C01814=1167.617,49.371,-49.076,-179.587,6.107,148.976
C01815=1167.621,49.121,-49.060,-179.589,6.107,148.977
C01816=1167.627,48.872,-49.044,-179.592,6.106,148.978
C01817=1167.632,48.622,-49.029,-179.594,6.104,148.978
C01818=1167.636,48.373,-49.012,-179.597,6.104,148.979
C01819=1167.641,48.124,-48.997,-179.599,6.103,148.979
C01820=1167.647,47.874,-48.981,-179.602,6.102,148.980
C01821=1167.652,47.624,-48.965,-179.605,6.101,148.980
C01822=1167.656,47.375,-48.950,-179.607,6.100,148.981
C01823=1167.662,47.126,-48.935,-179.610,6.099,148.982
C01824=1167.666,46.876,-48.919,-179.612,6.098,148.982
C01825=1167.671,46.627,-48.902,-179.615,6.098,148.983
C01826=1167.677,46.377,-48.887,-179.618,6.096,148.983
C01827=1167.681,46.128,-48.872,-179.621,6.096,148.984
C01828=1167.686,45.878,-48.856,-179.623,6.095,148.984
C01829=1167.692,45.629,-48.840,-179.626,6.093,148.985
C01830=1167.696,45.380,-48.825,-179.628,6.093,148.985
C01831=1167.702,45.130,-48.810,-179.631,6.092,148.986
C01832=1167.706,44.880,-48.794,-179.633,6.090,148.986
C01833=1167.712,44.631,-48.778,-179.636,6.090,148.987
C01834=1167.716,44.382,-48.763,-179.638,6.089,148.988
C01835=1167.721,44.132,-48.747,-179.641,6.088,148.988
C01836=1167.727,43.882,-48.732,-179.644,6.087,148.989
C01837=1167.731,43.633,-48.717,-179.646,6.086,148.989
C01838=1167.737,43.384,-48.701,-179.648,6.085,148.990
C01839=1167.742,43.134,-48.686,-179.652,6.084,148.990
C01840=1167.746,42.884,-48.670,-179.654,6.083,148.991
C01841=1167.752,42.635,-48.655,-179.656,6.083,148.992
C01842=1167.757,42.386,-48.639,-179.660,6.082,148.992
C01843=1167.762,42.137,-48.624,-179.662,6.081,148.993
C01844=1167.766,41.886,-48.608,-179.664,6.080,148.993
C01845=1167.771,41.637,-48.593,-179.667,6.079,148.994
C01846=1167.776,41.388,-48.577,-179.670,6.078,148.994
C01847=1167.782,41.139,-48.562,-179.672,6.077,148.995
C01848=1167.787,40.889,-48.548,-179.675,6.077,148.996
C01849=1167.792,40.639,-48.532,-179.677,6.075,148.996
C01850=1167.797,40.389,-48.516,-179.680,6.075,148.997
C01851=1167.802,40.140,-48.501,-179.682,6.074,148.997
C01852=1167.807,39.891,-48.485,-179.685,6.072,148.998
C01853=1167.812,39.642,-48.470,-179.688,6.072,148.998
C01854=1167.817,39.392,-48.455,-179.690,6.071,148.999
C01855=1167.822,39.143,-48.441,-179.693,6.071,149.000
C01856=1167.827,38.893,-48.425,-179.696,6.069,149.000
C01857=1167.832,38.643,-48.409,-179.698,6.068,149.001
C01858=1167.837,38.394,-48.394,-179.700,6.068,149.001
C01859=1167.842,38.145,-48.379,-179.703,6.067,149.002
C01860=1167.847,37.895,-48.364,-179.706,6.065,149.002
C01861=1167.852,37.646,-48.349,-179.708,6.065,149.003
C01862=1167.857,37.396,-48.334,-179.711,6.064,149.003
C01863=1167.862,37.146,-48.318,-179.714,6.063,149.004
C01864=1167.867,36.897,-48.303,-179.716,6.062,149.005
C01865=1167.872,36.647,-48.288,-179.719,6.061,149.005
C01866=1167.877,36.398,-48.273,-179.721,6.061,149.006
C01867=1167.882,36.149,-48.257,-179.724,6.059,149.006
C01868=1167.887,35.899,-48.243,-179.727,6.059,149.007
C01869=1167.893,35.650,-48.227,-179.729,6.058,149.007
C01870=1167.897,35.401,-48.212,-179.732,6.057,149.008
C01871=1167.903,35.151,-48.197,-179.734,6.056,149.009
C01872=1167.907,34.901,-48.182,-179.737,6.055,149.009
C01873=1167.912,34.651,-48.167,-179.739,6.054,149.010
C01874=1167.917,34.402,-48.152,-179.742,6.054,149.010
C01875=1167.922,34.153,-48.137,-179.745,6.053,149.011
C01876=1167.927,33.903,-48.122,-179.747,6.052,149.012
C01877=1167.932,33.653,-48.107,-179.750,6.051,149.012
C01878=1167.938,33.404,-48.092,-179.752,6.050,149.013
C01879=1167.942,33.155,-48.077,-179.755,6.049,149.013
C01880=1167.948,32.905,-48.062,-179.757,6.048,149.014
C01881=1167.953,32.656,-48.047,-179.760,6.048,149.014
C01882=1167.958,32.406,-48.033,-179.762,6.047,149.015
C01883=1167.963,32.157,-48.017,-179.765,6.046,149.016
C01884=1167.968,31.908,-48.002,-179.768,6.045,149.016
C01885=1167.973,31.658,-47.988,-179.770,6.044,149.017
C01886=1167.978,31.408,-47.972,-179.773,6.044,149.017
C01887=1167.983,31.159,-47.958,-179.775,6.043,149.018
C01888=1167.988,30.909,-47.942,-179.778,6.042,149.018
C01889=1167.993,30.660,-47.928,-179.780,6.041,149.019
C01890=1167.998,30.411,-47.913,-179.783,6.040,149.020
C01891=1168.004,30.161,-47.898,-179.785,6.040,149.020
C01892=1168.008,29.911,-47.883,-179.788,6.038,149.021
C01893=1168.013,29.662,-47.869,-179.791,6.038,149.021
C01894=1168.019,29.412,-47.853,-179.793,6.037,149.022
C01895=1168.024,29.163,-47.839,-179.796,6.036,149.023
C01896=1168.028,28.914,-47.824,-179.798,6.036,149.023
C01897=1168.033,28.664,-47.810,-179.801,6.034,149.024
C01898=1168.039,28.395,-47.794,-179.804,6.034,149.024
C01899=1168.044,28.126,-47.778,-179.806,6.033,149.025
C01900=1168.050,27.857,-47.762,-179.809,6.032,149.025
C01901=1168.055,27.588,-47.746,-179.812,6.031,149.026
C01902=1168.060,27.339,-47.731,-179.814,6.030,149.027
C01903=1168.065,27.089,-47.717,-179.817,6.029,149.027
C01904=1168.071,26.839,-47.702,-179.820,6.029,149.028
C01905=1168.075,26.590,-47.687,-179.822,6.028,149.028
C01906=1168.080,26.340,-47.672,-179.825,6.027,149.029
C01907=1168.085,26.091,-47.657,-179.827,6.026,149.030
C01908=1168.090,25.841,-47.643,-179.830,6.025,149.030
C01909=1168.095,25.592,-47.628,-179.832,6.024,149.031
C01910=1168.100,25.342,-47.613,-179.835,6.024,149.031
C01911=1168.105,25.093,-47.599,-179.838,6.023,149.032
C01912=1168.111,24.843,-47.584,-179.840,6.023,149.033
C01913=1168.116,24.594,-47.570,-179.843,6.021,149.033
C01914=1168.121,24.345,-47.555,-179.845,6.020,149.034
C01915=1168.126,24.095,-47.541,-179.848,6.020,149.034
C01916=1168.131,23.845,-47.527,-179.850,6.019,149.035
C01917=1168.135,23.596,-47.512,-179.853,6.019,149.035
C01918=1168.141,23.346,-47.497,-179.856,6.017,149.036
C01919=1168.146,23.096,-47.483,-179.858,6.016,149.037
C01920=1168.151,22.847,-47.468,-179.861,6.016,149.037
C01921=1168.156,22.598,-47.453,-179.863,6.015,149.038
C01922=1168.161,22.348,-47.439,-179.866,6.015,149.038
C01923=1168.166,22.099,-47.425,-179.868,6.014,149.039
C01924=1168.171,21.849,-47.411,-179.871,6.013,149.040
C01925=1168.177,21.600,-47.395,-179.874,6.012,149.040
C01926=1168.182,21.350,-47.381,-179.876,6.011,149.041
C01927=1168.186,21.100,-47.367,-179.878,6.011,149.041
C01928=1168.191,20.851,-47.352,-179.881,6.010,149.042
C01929=1168.196,20.601,-47.338,-179.883,6.009,149.042
C01930=1168.201,20.351,-47.324,-179.886,6.008,149.043
C01931=1168.207,20.103,-47.309,-179.889,6.007,149.044
C01932=1168.212,19.853,-47.295,-179.891,6.007,149.044
C01933=1168.217,19.603,-47.281,-179.893,6.006,149.045
C01934=1168.221,19.354,-47.266,-179.896,6.006,149.045
C01935=1168.227,19.104,-47.251,-179.898,6.005,149.046
C01936=1168.232,18.854,-47.237,-179.901,6.003,149.047
C01937=1168.238,18.605,-47.223,-179.904,6.003,149.047
C01938=1168.243,18.355,-47.209,-179.906,6.002,149.048
C01939=1168.247,18.106,-47.194,-179.909,6.002,149.048
C01940=1168.252,17.856,-47.180,-179.911,6.001,149.049
C01941=1168.257,17.607,-47.165,-179.914,6.000,149.050
C01942=1168.263,17.358,-47.152,-179.916,6.000,149.050
C01943=1168.268,17.108,-47.137,-179.919,5.998,149.051
C01944=1168.273,16.858,-47.123,-179.922,5.998,149.051
C01945=1168.278,16.609,-47.109,-179.924,5.997,149.052
C01946=1168.283,16.359,-47.094,-179.927,5.996,149.052
C01947=1168.288,16.110,-47.081,-179.929,5.996,149.053
C01948=1168.293,15.860,-47.066,-179.931,5.995,149.054
C01949=1168.298,15.610,-47.052,-179.934,5.995,149.054
C01950=1168.303,15.361,-47.038,-179.937,5.993,149.055
C01951=1168.309,15.112,-47.024,-179.940,5.992,149.055
C01952=1168.313,14.862,-47.010,-179.942,5.992,149.056
C01953=1168.318,14.612,-46.995,-179.944,5.991,149.057
C01954=1168.323,14.363,-46.981,-179.947,5.991,149.057
C01955=1168.329,14.114,-46.967,-179.949,5.990,149.058
C01956=1168.333,13.864,-46.953,-179.952,5.989,149.058
C01957=1168.338,13.614,-46.939,-179.955,5.988,149.059
C01958=1168.343,13.365,-46.925,-179.957,5.987,149.060
C01959=1168.349,13.115,-46.912,-179.960,5.987,149.060
C01960=1168.354,12.865,-46.897,-179.962,5.986,149.061
C01961=1168.359,12.616,-46.883,-179.965,5.986,149.061
C01962=1168.364,12.366,-46.869,-179.967,5.985,149.062
C01963=1168.369,12.117,-46.855,-179.969,5.984,149.063
C01964=1168.374,11.867,-46.841,-179.972,5.984,149.063
C01965=1168.379,11.618,-46.826,-179.974,5.983,149.064
C01966=1168.384,11.369,-46.813,-179.978,5.982,149.064
C01967=1168.389,11.119,-46.799,-179.980,5.981,149.065
C01968=1168.394,10.869,-46.785,-179.982,5.980,149.065
C01969=1168.399,10.619,-46.771,-179.985,5.979,149.066
C01970=1168.405,10.370,-46.757,-179.987,5.979,149.067
C01971=1168.410,10.120,-46.743,-179.990,5.979,149.067
C01972=1168.415,9.871,-46.728,-179.992,5.978,149.068
C01973=1168.420,9.621,-46.716,-179.995,5.977,149.068
C01974=1168.425,9.372,-46.702,-179.997,5.976,149.069
C01975=1168.430,9.122,-46.687,180.000,5.975,149.070
C01976=1168.435,8.873,-46.673,179.997,5.975,149.070
C01977=1168.441,8.623,-46.660,179.995,5.974,149.071
C01978=1168.446,8.373,-46.646,179.992,5.973,149.071
C01979=1168.450,8.124,-46.632,179.990,5.973,149.072
C01980=1168.455,7.875,-46.618,179.988,5.972,149.073
C01981=1168.461,7.624,-46.604,179.985,5.972,149.073
C01982=1168.466,7.375,-46.590,179.983,5.971,149.074
C01983=1168.470,7.126,-46.577,179.980,5.970,149.074
C01984=1168.476,6.877,-46.563,179.978,5.969,149.075
C01985=1168.481,6.626,-46.549,179.975,5.969,149.076
C01986=1168.486,6.377,-46.535,179.972,5.968,149.076
C01987=1168.491,6.128,-46.522,179.970,5.967,149.077
C01988=1168.496,5.878,-46.508,179.967,5.966,149.077
C01989=1168.501,5.628,-46.494,179.965,5.966,149.078
C01990=1168.507,5.379,-46.480,179.962,5.965,149.079
C01991=1168.511,5.129,-46.467,179.960,5.965,149.079
C01992=1168.517,4.880,-46.453,179.958,5.964,149.080
C01993=1168.522,4.630,-46.440,179.955,5.963,149.080
C01994=1168.527,4.380,-46.425,179.953,5.963,149.081
C01995=1168.532,4.131,-46.412,179.950,5.962,149.082
C01996=1168.537,3.881,-46.398,179.947,5.962,149.082
C01997=1168.543,3.632,-46.384,179.945,5.961,149.083
C01998=1168.547,3.382,-46.371,179.943,5.960,149.083
C01999=1168.553,3.133,-46.358,179.941,5.960,149.084
C02000=1168.558,2.883,-46.343,179.937,5.958,149.085
C02001=1168.562,2.633,-46.330,179.935,5.958,149.085
C02002=1168.568,2.364,-46.316,179.932,5.957,149.086
C02003=1168.574,2.095,-46.301,179.930,5.956,149.086
C02004=1168.579,1.826,-46.286,179.927,5.956,149.087
C02005=1168.585,1.556,-46.271,179.924,5.956,149.088
C02006=1168.590,1.307,-46.258,179.921,5.954,149.088
C02007=1168.595,1.056,-46.245,179.919,5.953,149.089
C02008=1168.600,0.808,-46.231,179.916,5.953,149.090
C02009=1168.605,0.557,-46.218,179.914,5.952,149.090
C02010=1168.611,0.308,-46.204,179.912,5.952,149.091
C02011=1168.615,0.058,-46.191,179.909,5.951,149.091
C02012=1168.621,-0.191,-46.177,179.907,5.950,149.092
C02013=1168.626,-0.441,-46.163,179.904,5.950,149.093
C02014=1168.631,-0.690,-46.150,179.902,5.949,149.093
C02015=1168.636,-0.940,-46.136,179.899,5.949,149.094
C02016=1168.641,-1.189,-46.123,179.897,5.948,149.094
C02017=1168.646,-1.439,-46.110,179.894,5.947,149.095
C02018=1168.651,-1.688,-46.097,179.892,5.947,149.096
C02019=1168.656,-1.938,-46.083,179.890,5.946,149.096
C02020=1168.662,-2.188,-46.070,179.887,5.946,149.097
C02021=1168.666,-2.437,-46.056,179.884,5.945,149.097
C02022=1168.672,-2.687,-46.043,179.882,5.944,149.098
C02023=1168.677,-2.937,-46.030,179.879,5.944,149.099
C02024=1168.682,-3.186,-46.016,179.877,5.943,149.099
C02025=1168.687,-3.436,-46.003,179.875,5.943,149.100
C02026=1168.693,-3.685,-45.990,179.872,5.942,149.100
C02027=1168.697,-3.935,-45.976,179.870,5.941,149.101
C02028=1168.703,-4.184,-45.963,179.867,5.941,149.102
C02029=1168.707,-4.434,-45.950,179.865,5.940,149.102
C02030=1168.713,-4.683,-45.936,179.862,5.940,149.103
C02031=1168.717,-4.933,-45.923,179.860,5.939,149.103
C02032=1168.723,-5.183,-45.910,179.858,5.938,149.104
C02033=1168.728,-5.432,-45.896,179.854,5.937,149.105
C02034=1168.733,-5.682,-45.883,179.852,5.937,149.105
C02035=1168.738,-5.931,-45.870,179.849,5.936,149.106
C02036=1168.744,-6.182,-45.857,179.847,5.935,149.106
C02037=1168.748,-6.430,-45.843,179.845,5.935,149.107
C02038=1168.753,-6.680,-45.830,179.842,5.934,149.108
C02039=1168.759,-6.930,-45.817,179.839,5.934,149.108
C02040=1168.764,-7.179,-45.805,179.837,5.933,149.109
C02041=1168.769,-7.429,-45.790,179.834,5.932,149.109
C02042=1168.774,-7.678,-45.778,179.832,5.932,149.110
C02043=1168.779,-7.929,-45.764,179.830,5.931,149.111
C02044=1168.784,-8.178,-45.752,179.827,5.931,149.111
C02045=1168.789,-8.427,-45.739,179.825,5.930,149.112
C02046=1168.794,-8.677,-45.725,179.822,5.929,149.112
C02047=1168.800,-8.926,-45.712,179.820,5.929,149.113
C02048=1168.805,-9.177,-45.698,179.817,5.928,149.114
C02049=1168.810,-9.426,-45.686,179.815,5.928,149.114
C02050=1168.815,-9.675,-45.673,179.812,5.927,149.115
C02051=1168.820,-9.926,-45.660,179.810,5.926,149.115
C02052=1168.825,-10.175,-45.647,179.808,5.926,149.116
C02053=1168.830,-10.424,-45.634,179.805,5.925,149.117
C02054=1168.835,-10.674,-45.620,179.802,5.925,149.117
C02055=1168.841,-10.923,-45.608,179.800,5.924,149.118
C02056=1168.845,-11.173,-45.595,179.797,5.923,149.118
C02057=1168.851,-11.423,-45.581,179.795,5.923,149.119
C02058=1168.856,-11.672,-45.569,179.793,5.922,149.120
C02059=1168.861,-11.922,-45.556,179.790,5.922,149.120
C02060=1168.867,-12.172,-45.543,179.788,5.922,149.121
C02061=1168.872,-12.421,-45.530,179.786,5.921,149.121
C02062=1168.876,-12.671,-45.517,179.783,5.921,149.122
C02063=1168.882,-12.921,-45.504,179.781,5.920,149.123
C02064=1168.887,-13.170,-45.491,179.778,5.919,149.123
C02065=1168.892,-13.420,-45.478,179.776,5.919,149.124
C02066=1168.898,-13.670,-45.465,179.773,5.918,149.124
C02067=1168.902,-13.919,-45.452,179.771,5.918,149.125
C02068=1168.907,-14.168,-45.439,179.769,5.917,149.126
C02069=1168.912,-14.418,-45.426,179.766,5.916,149.126
C02070=1168.918,-14.668,-45.414,179.764,5.916,149.127
C02071=1168.923,-14.917,-45.401,179.761,5.915,149.127
C02072=1168.928,-15.167,-45.388,179.758,5.915,149.128
C02073=1168.933,-15.417,-45.376,179.756,5.914,149.129
C02074=1168.939,-15.666,-45.362,179.754,5.913,149.129
C02075=1168.944,-15.916,-45.350,179.751,5.913,149.130
C02076=1168.948,-16.166,-45.337,179.749,5.912,149.130
C02077=1168.954,-16.415,-45.324,179.746,5.912,149.131
C02078=1168.959,-16.665,-45.311,179.744,5.911,149.132
C02079=1168.964,-16.915,-45.298,179.741,5.911,149.132
C02080=1168.969,-17.164,-45.286,179.739,5.910,149.133
C02081=1168.974,-17.413,-45.273,179.736,5.909,149.133
C02082=1168.979,-17.663,-45.260,179.734,5.909,149.134
C02083=1168.985,-17.913,-45.247,179.732,5.908,149.135
C02084=1168.990,-18.163,-45.235,179.729,5.908,149.135
C02085=1168.995,-18.412,-45.222,179.726,5.907,149.136
C02086=1169.000,-18.662,-45.210,179.724,5.906,149.136
C02087=1169.005,-18.911,-45.197,179.722,5.907,149.137
C02088=1169.010,-19.161,-45.184,179.720,5.906,149.138
C02089=1169.016,-19.411,-45.171,179.717,5.905,149.138
C02090=1169.021,-19.660,-45.158,179.715,5.905,149.139
C02091=1169.026,-19.910,-45.146,179.712,5.904,149.140
C02092=1169.031,-20.160,-45.133,179.710,5.904,149.140
C02093=1169.036,-20.409,-45.121,179.707,5.903,149.141
C02094=1169.041,-20.658,-45.108,179.705,5.902,149.141
C02095=1169.046,-20.908,-45.096,179.702,5.902,149.142
C02096=1169.052,-21.158,-45.083,179.700,5.901,149.143
C02097=1169.057,-21.408,-45.070,179.697,5.901,149.143
C02098=1169.062,-21.657,-45.058,179.695,5.900,149.144
C02099=1169.067,-21.907,-45.045,179.693,5.899,149.144
C02100=1169.073,-22.157,-45.033,179.690,5.899,149.145
C02101=1169.078,-22.406,-45.021,179.688,5.898,149.146
C02102=1169.083,-22.655,-45.008,179.686,5.899,149.146
C02103=1169.087,-22.905,-44.995,179.683,5.898,149.147
C02104=1169.093,-23.155,-44.983,179.681,5.897,149.147
C02105=1169.098,-23.405,-44.970,179.678,5.897,149.148
C02106=1169.104,-23.675,-44.956,179.675,5.896,149.149
C02107=1169.110,-23.944,-44.944,179.673,5.896,149.149
C02108=1169.115,-24.214,-44.930,179.671,5.895,149.150
C02109=1169.121,-24.485,-44.916,179.667,5.894,149.151
C02110=1169.126,-24.734,-44.904,179.665,5.894,149.151
C02111=1169.131,-24.983,-44.891,179.663,5.893,149.152
C02112=1169.136,-25.233,-44.879,179.660,5.893,149.153
C02113=1169.141,-25.482,-44.867,179.658,5.893,149.153
C02114=1169.147,-25.732,-44.854,179.656,5.892,149.154
C02115=1169.152,-25.982,-44.842,179.653,5.891,149.154
C02116=1169.157,-26.231,-44.830,179.651,5.891,149.155
C02117=1169.162,-26.482,-44.817,179.648,5.890,149.156
C02118=1169.167,-26.731,-44.805,179.645,5.890,149.156
C02119=1169.172,-26.980,-44.792,179.643,5.889,149.157
C02120=1169.178,-27.230,-44.780,179.641,5.888,149.157
C02121=1169.183,-27.480,-44.768,179.639,5.888,149.158
C02122=1169.188,-27.730,-44.756,179.636,5.888,149.159
C02123=1169.193,-27.979,-44.743,179.634,5.888,149.159
C02124=1169.198,-28.228,-44.731,179.632,5.887,149.160
C02125=1169.203,-28.478,-44.719,179.629,5.886,149.160
C02126=1169.208,-28.728,-44.706,179.627,5.885,149.161
C02127=1169.213,-28.978,-44.694,179.624,5.885,149.162
C02128=1169.218,-29.227,-44.682,179.621,5.885,149.162
C02129=1169.224,-29.477,-44.670,179.619,5.884,149.163
C02130=1169.229,-29.726,-44.657,179.617,5.883,149.164
C02131=1169.234,-29.976,-44.645,179.615,5.883,149.164
C02132=1169.239,-30.226,-44.633,179.612,5.883,149.165
C02133=1169.245,-30.476,-44.621,179.610,5.882,149.165
C02134=1169.250,-30.725,-44.608,179.607,5.882,149.166
C02135=1169.255,-30.975,-44.596,179.605,5.881,149.167
C02136=1169.260,-31.224,-44.584,179.603,5.880,149.167
C02137=1169.265,-31.474,-44.573,179.600,5.880,149.168
C02138=1169.270,-31.724,-44.561,179.597,5.880,149.168
C02139=1169.276,-31.973,-44.548,179.596,5.880,149.169
C02140=1169.281,-32.223,-44.536,179.593,5.879,149.170
C02141=1169.286,-32.472,-44.524,179.591,5.878,149.170
C02142=1169.292,-32.722,-44.512,179.588,5.878,149.171
C02143=1169.297,-32.971,-44.499,179.586,5.877,149.171
C02144=1169.301,-33.221,-44.488,179.583,5.877,149.172
C02145=1169.307,-33.471,-44.476,179.581,5.876,149.173
C02146=1169.312,-33.720,-44.463,179.578,5.876,149.173
C02147=1169.317,-33.970,-44.451,179.576,5.876,149.174
C02148=1169.323,-34.220,-44.440,179.574,5.875,149.174
C02149=1169.328,-34.470,-44.427,179.572,5.874,149.175
C02150=1169.333,-34.719,-44.416,179.569,5.874,149.176
C02151=1169.338,-34.968,-44.403,179.566,5.874,149.176
C02152=1169.343,-35.218,-44.391,179.564,5.873,149.177
C02153=1169.349,-35.468,-44.379,179.561,5.872,149.178
C02154=1169.354,-35.718,-44.367,179.560,5.872,149.178
C02155=1169.358,-35.967,-44.355,179.557,5.872,149.179
C02156=1169.364,-36.217,-44.344,179.554,5.872,149.179
C02157=1169.369,-36.467,-44.332,179.552,5.871,149.180
C02158=1169.374,-36.716,-44.319,179.550,5.870,149.181
C02159=1169.380,-36.966,-44.307,179.547,5.869,149.181
C02160=1169.385,-37.216,-44.296,179.545,5.869,149.182
C02161=1169.390,-37.465,-44.283,179.543,5.869,149.182
C02162=1169.395,-37.715,-44.271,179.541,5.869,149.183
C02163=1169.401,-37.965,-44.260,179.538,5.868,149.184
C02164=1169.405,-38.215,-44.248,179.536,5.867,149.184
C02165=1169.410,-38.464,-44.236,179.533,5.867,149.185
C02166=1169.416,-38.714,-44.224,179.530,5.867,149.185
C02167=1169.420,-38.964,-44.212,179.528,5.866,149.186
C02168=1169.426,-39.214,-44.201,179.526,5.866,149.187
C02169=1169.431,-39.464,-44.189,179.524,5.865,149.187
C02170=1169.437,-39.712,-44.176,179.521,5.865,149.188
C02171=1169.442,-39.962,-44.165,179.519,5.864,149.188
C02172=1169.447,-40.212,-44.153,179.516,5.864,149.189
C02173=1169.453,-40.462,-44.141,179.514,5.863,149.190
C02174=1169.457,-40.711,-44.130,179.512,5.863,149.190
C02175=1169.463,-40.961,-44.118,179.509,5.863,149.191
C02176=1169.468,-41.211,-44.106,179.507,5.862,149.191
C02177=1169.473,-41.460,-44.094,179.505,5.862,149.192
C02178=1169.478,-41.710,-44.082,179.502,5.861,149.193
C02179=1169.483,-41.960,-44.071,179.500,5.860,149.193
C02180=1169.489,-42.209,-44.060,179.498,5.861,149.194
C02181=1169.494,-42.459,-44.048,179.496,5.860,149.194
C02182=1169.500,-42.709,-44.036,179.493,5.859,149.195
C02183=1169.504,-42.959,-44.025,179.490,5.859,149.196
C02184=1169.509,-43.208,-44.012,179.488,5.858,149.196
C02185=1169.514,-43.457,-44.001,179.486,5.859,149.197
C02186=1169.519,-43.707,-43.989,179.484,5.858,149.197
C02187=1169.525,-43.957,-43.977,179.481,5.857,149.198
C02188=1169.530,-44.206,-43.966,179.478,5.857,149.199
C02189=1169.536,-44.456,-43.954,179.476,5.856,149.199
C02190=1169.541,-44.706,-43.942,179.474,5.856,149.200
C02191=1169.546,-44.956,-43.931,179.472,5.856,149.201
C02192=1169.551,-45.206,-43.919,179.469,5.855,149.201
C02193=1169.556,-45.455,-43.908,179.467,5.855,149.202
C02194=1169.562,-45.705,-43.896,179.464,5.854,149.202
C02195=1169.567,-45.954,-43.885,179.462,5.854,149.203
C02196=1169.572,-46.204,-43.873,179.460,5.854,149.204
C02197=1169.577,-46.454,-43.861,179.458,5.853,149.204
C02198=1169.582,-46.704,-43.850,179.455,5.852,149.205
C02199=1169.588,-46.954,-43.838,179.453,5.852,149.205
C02200=1169.593,-47.203,-43.827,179.450,5.852,149.206
C02201=1169.598,-47.452,-43.815,179.448,5.852,149.207
C02202=1169.603,-47.702,-43.804,179.446,5.851,149.207
C02203=1169.608,-47.952,-43.792,179.444,5.850,149.208
C02204=1169.613,-48.202,-43.781,179.441,5.850,149.209
C02205=1169.619,-48.451,-43.769,179.438,5.849,149.209
C02206=1169.624,-48.701,-43.758,179.437,5.849,149.210
C02207=1169.629,-48.950,-43.746,179.434,5.849,149.210
C02208=1169.634,-49.201,-43.735,179.432,5.848,149.211
C02209=1169.640,-49.451,-43.724,179.429,5.848,149.212
C02210=1169.646,-49.720,-43.711,179.427,5.847,149.212
C02211=1169.651,-49.991,-43.699,179.424,5.847,149.213
C02212=1169.657,-50.261,-43.686,179.422,5.846,149.213
C02213=1169.662,-50.532,-43.674,179.419,5.846,149.214
C02214=1169.667,-50.782,-43.663,179.417,5.846,149.215
C02215=1169.672,-51.031,-43.651,179.415,5.845,149.215
C02216=1169.678,-51.280,-43.640,179.412,5.845,149.216
C02217=1169.683,-51.531,-43.629,179.410,5.844,149.217
C02218=1169.689,-51.781,-43.617,179.407,5.844,149.217
C02219=1169.693,-52.030,-43.606,179.405,5.844,149.218
C02220=1169.699,-52.279,-43.594,179.403,5.843,149.218
C02221=1169.704,-52.529,-43.583,179.400,5.843,149.219
C02222=1169.709,-52.779,-43.572,179.398,5.842,149.220
C02223=1169.715,-53.029,-43.561,179.396,5.842,149.220
C02224=1169.720,-53.278,-43.550,179.394,5.842,149.221
C02225=1169.725,-53.528,-43.538,179.391,5.841,149.221
C02226=1169.730,-53.778,-43.527,179.388,5.841,149.222
C02227=1169.735,-54.027,-43.516,179.387,5.841,149.223
C02228=1169.741,-54.277,-43.505,179.384,5.840,149.223
C02229=1169.746,-54.527,-43.493,179.382,5.840,149.224
C02230=1169.751,-54.777,-43.481,179.379,5.839,149.225
C02231=1169.757,-55.026,-43.471,179.377,5.838,149.225
C02232=1169.761,-55.276,-43.460,179.375,5.839,149.226
C02233=1169.767,-55.526,-43.448,179.372,5.838,149.226
C02234=1169.772,-55.775,-43.437,179.370,5.838,149.227
C02235=1169.777,-56.025,-43.426,179.368,5.837,149.228
C02236=1169.782,-56.275,-43.415,179.366,5.837,149.228
C02237=1169.788,-56.524,-43.404,179.363,5.837,149.229
C02238=1169.793,-56.774,-43.393,179.361,5.836,149.229
C02239=1169.798,-57.024,-43.381,179.358,5.836,149.230
C02240=1169.803,-57.273,-43.370,179.356,5.836,149.231
C02241=1169.808,-57.523,-43.360,179.354,5.835,149.231
C02242=1169.814,-57.773,-43.348,179.352,5.835,149.232
C02243=1169.819,-58.022,-43.337,179.349,5.834,149.232
C02244=1169.824,-58.272,-43.326,179.347,5.834,149.233
C02245=1169.829,-58.522,-43.315,179.345,5.834,149.234
C02246=1169.835,-58.771,-43.304,179.342,5.833,149.234
C02247=1169.840,-59.021,-43.293,179.340,5.833,149.235
C02248=1169.845,-59.271,-43.282,179.338,5.833,149.235
C02249=1169.851,-59.520,-43.270,179.336,5.832,149.236
C02250=1169.856,-59.771,-43.260,179.333,5.831,149.237
C02251=1169.860,-60.020,-43.248,179.331,5.831,149.237
C02252=1169.866,-60.270,-43.238,179.329,5.831,149.238
C02253=1169.871,-60.520,-43.226,179.326,5.831,149.238
C02254=1169.876,-60.770,-43.216,179.324,5.830,149.239
C02255=1169.882,-61.019,-43.205,179.322,5.829,149.240
C02256=1169.886,-61.268,-43.193,179.319,5.830,149.240
C02257=1169.893,-61.518,-43.183,179.317,5.829,149.241
C02258=1169.897,-61.768,-43.171,179.315,5.829,149.242
C02259=1169.902,-62.018,-43.161,179.312,5.828,149.242
C02260=1169.908,-62.267,-43.150,179.310,5.828,149.243
C02261=1169.913,-62.517,-43.139,179.308,5.827,149.243
C02262=1169.919,-62.767,-43.128,179.306,5.827,149.244
C02263=1169.924,-63.017,-43.117,179.303,5.827,149.245
C02264=1169.928,-63.266,-43.106,179.301,5.827,149.245
C02265=1169.934,-63.516,-43.096,179.299,5.826,149.246
C02266=1169.939,-63.766,-43.084,179.296,5.825,149.246
C02267=1169.945,-64.016,-43.074,179.294,5.826,149.247
C02268=1169.950,-64.265,-43.062,179.292,5.825,149.247
C02269=1169.955,-64.515,-43.052,179.289,5.825,149.248
C02270=1169.960,-64.764,-43.041,179.287,5.824,149.249
C02271=1169.965,-65.015,-43.030,179.285,5.824,149.249
C02272=1169.971,-65.264,-43.020,179.283,5.823,149.250
C02273=1169.976,-65.514,-43.008,179.280,5.823,149.251
C02274=1169.982,-65.764,-42.998,179.278,5.823,149.251
C02275=1169.986,-66.013,-42.987,179.276,5.823,149.252
C02276=1169.992,-66.263,-42.976,179.273,5.822,149.252
C02277=1169.997,-66.512,-42.965,179.271,5.821,149.253
C02278=1170.002,-66.762,-42.955,179.269,5.822,149.254
C02279=1170.007,-67.012,-42.944,179.267,5.821,149.254
C02280=1170.013,-67.261,-42.933,179.264,5.821,149.255
C02281=1170.018,-67.512,-42.922,179.263,5.821,149.255
C02282=1170.024,-67.761,-42.912,179.260,5.820,149.256
C02283=1170.028,-68.011,-42.901,179.257,5.820,149.257
C02284=1170.034,-68.260,-42.891,179.255,5.819,149.257
C02285=1170.039,-68.510,-42.879,179.253,5.819,149.258
C02286=1170.044,-68.760,-42.869,179.251,5.819,149.258
C02287=1170.049,-69.010,-42.858,179.248,5.818,149.259
C02288=1170.055,-69.259,-42.848,179.247,5.818,149.260
C02289=1170.060,-69.509,-42.837,179.244,5.818,149.260
C02290=1170.065,-69.758,-42.827,179.242,5.817,149.261
C02291=1170.070,-70.009,-42.816,179.240,5.817,149.261
C02292=1170.076,-70.258,-42.805,179.238,5.817,149.262
C02293=1170.081,-70.508,-42.794,179.235,5.816,149.263
C02294=1170.087,-70.758,-42.784,179.233,5.815,149.263
C02295=1170.092,-71.007,-42.773,179.231,5.816,149.264
C02296=1170.097,-71.257,-42.762,179.228,5.815,149.265
C02297=1170.102,-71.507,-42.752,179.226,5.815,149.265
C02298=1170.108,-71.757,-42.742,179.224,5.815,149.266
C02299=1170.112,-72.006,-42.730,179.221,5.814,149.266
C02300=1170.118,-72.256,-42.720,179.219,5.814,149.267
C02301=1170.123,-72.506,-42.709,179.217,5.814,149.267
C02302=1170.129,-72.756,-42.699,179.215,5.813,149.268
C02303=1170.134,-73.005,-42.688,179.212,5.813,149.269
C02304=1170.139,-73.255,-42.678,179.210,5.813,149.269
C02305=1170.145,-73.504,-42.668,179.208,5.812,149.270
C02306=1170.150,-73.755,-42.657,179.205,5.812,149.270
C02307=1170.155,-74.004,-42.647,179.203,5.811,149.271
C02308=1170.160,-74.254,-42.636,179.201,5.811,149.272
C02309=1170.165,-74.503,-42.625,179.199,5.811,149.272
C02310=1170.171,-74.753,-42.615,179.196,5.810,149.273
C02311=1170.176,-75.003,-42.605,179.195,5.810,149.273
C02312=1170.182,-75.253,-42.594,179.192,5.810,149.274
C02313=1170.187,-75.503,-42.584,179.189,5.809,149.275
C02314=1170.192,-75.773,-42.573,179.188,5.809,149.275
C02315=1170.198,-76.044,-42.561,179.185,5.809,149.276
C02316=1170.203,-76.316,-42.550,179.182,5.809,149.277
C02317=1170.210,-76.587,-42.539,179.180,5.808,149.277
C02318=1170.215,-76.837,-42.528,179.178,5.807,149.278
C02319=1170.220,-77.086,-42.518,179.176,5.807,149.278
C02320=1170.225,-77.337,-42.507,179.173,5.807,149.279
C02321=1170.231,-77.586,-42.497,179.171,5.807,149.280
C02322=1170.236,-77.835,-42.486,179.169,5.807,149.280
C02323=1170.240,-78.085,-42.476,179.166,5.806,149.281
C02324=1170.246,-78.335,-42.466,179.164,5.806,149.281
C02325=1170.252,-78.584,-42.456,179.162,5.806,149.282
C02326=1170.257,-78.834,-42.445,179.160,5.805,149.283
C02327=1170.262,-79.084,-42.435,179.158,5.806,149.283
C02328=1170.268,-79.334,-42.425,179.156,5.805,149.284
C02329=1170.273,-79.584,-42.414,179.153,5.804,149.285
C02330=1170.278,-79.833,-42.404,179.151,5.804,149.285
C02331=1170.283,-80.083,-42.394,179.149,5.804,149.286
C02332=1170.288,-80.333,-42.384,179.146,5.803,149.286
C02333=1170.294,-80.582,-42.374,179.144,5.804,149.287
C02334=1170.299,-80.833,-42.363,179.142,5.803,149.287
C02335=1170.304,-81.082,-42.353,179.140,5.802,149.288
C02336=1170.310,-81.332,-42.343,179.138,5.802,149.289
C02337=1170.314,-81.582,-42.333,179.135,5.802,149.289
C02338=1170.320,-81.831,-42.323,179.133,5.801,149.290
C02339=1170.326,-82.081,-42.312,179.131,5.802,149.290
C02340=1170.331,-82.331,-42.302,179.129,5.801,149.291
C02341=1170.336,-82.580,-42.292,179.126,5.800,149.292
C02342=1170.342,-82.830,-42.281,179.125,5.800,149.292
C02343=1170.347,-83.079,-42.272,179.122,5.800,149.293
C02344=1170.352,-83.329,-42.261,179.120,5.799,149.293
C02345=1170.358,-83.580,-42.252,179.118,5.800,149.294
C02346=1170.363,-83.829,-42.241,179.115,5.799,149.295
C02347=1170.367,-84.079,-42.231,179.113,5.799,149.295
C02348=1170.373,-84.329,-42.221,179.111,5.799,149.296
C02349=1170.379,-84.578,-42.211,179.108,5.798,149.296
C02350=1170.384,-84.828,-42.200,179.107,5.798,149.297
C02351=1170.388,-85.078,-42.191,179.104,5.798,149.298
C02352=1170.394,-85.327,-42.181,179.102,5.797,149.298
C02353=1170.400,-85.577,-42.170,179.100,5.797,149.299
C02354=1170.405,-85.828,-42.161,179.098,5.797,149.299
C02355=1170.410,-86.077,-42.151,179.095,5.796,149.300
C02356=1170.415,-86.326,-42.141,179.093,5.796,149.300
C02357=1170.420,-86.577,-42.130,179.091,5.796,149.301
C02358=1170.426,-86.826,-42.120,179.089,5.796,149.302
C02359=1170.431,-87.075,-42.110,179.087,5.795,149.302
C02360=1170.436,-87.325,-42.100,179.084,5.795,149.303
C02361=1170.442,-87.576,-42.090,179.082,5.795,149.304
C02362=1170.447,-87.825,-42.081,179.080,5.794,149.304
C02363=1170.452,-88.075,-42.070,179.077,5.794,149.305
C02364=1170.458,-88.324,-42.060,179.076,5.794,149.305
C02365=1170.462,-88.574,-42.050,179.074,5.793,149.306
C02366=1170.468,-88.824,-42.041,179.072,5.794,149.306
C02367=1170.474,-89.074,-42.031,179.069,5.793,149.307
C02368=1170.478,-89.323,-42.021,179.067,5.792,149.308
C02369=1170.484,-89.573,-42.011,179.065,5.792,149.308
C02370=1170.489,-89.823,-42.001,179.062,5.792,149.309
C02371=1170.494,-90.073,-41.991,179.060,5.791,149.309
C02372=1170.500,-90.322,-41.981,179.058,5.792,149.310
C02373=1170.505,-90.572,-41.971,179.056,5.791,149.311
C02374=1170.510,-90.822,-41.962,179.054,5.791,149.311
C02375=1170.516,-91.072,-41.951,179.052,5.790,149.312
C02376=1170.521,-91.321,-41.941,179.049,5.790,149.312
C02377=1170.526,-91.571,-41.932,179.047,5.790,149.313
C02378=1170.532,-91.821,-41.922,179.045,5.790,149.314
C02379=1170.537,-92.071,-41.912,179.043,5.790,149.314
C02380=1170.542,-92.321,-41.903,179.040,5.789,149.315
C02381=1170.548,-92.570,-41.892,179.038,5.789,149.315
C02382=1170.553,-92.820,-41.883,179.036,5.789,149.316
C02383=1170.558,-93.070,-41.873,179.034,5.788,149.316
C02384=1170.564,-93.319,-41.863,179.032,5.788,149.317
C02385=1170.568,-93.569,-41.853,179.030,5.788,149.318
C02386=1170.574,-93.819,-41.844,179.028,5.787,149.318
C02387=1170.579,-94.069,-41.834,179.025,5.787,149.319
C02388=1170.585,-94.318,-41.824,179.023,5.787,149.319
C02389=1170.590,-94.568,-41.815,179.021,5.787,149.320
C02390=1170.595,-94.818,-41.805,179.019,5.786,149.321
C02391=1170.601,-95.069,-41.795,179.016,5.786,149.321
C02392=1170.606,-95.318,-41.785,179.015,5.786,149.322
C02393=1170.611,-95.567,-41.775,179.012,5.786,149.322
C02394=1170.616,-95.817,-41.766,179.010,5.786,149.323
C02395=1170.622,-96.067,-41.756,179.008,5.785,149.323
C02396=1170.627,-96.317,-41.747,179.006,5.784,149.324
C02397=1170.633,-96.566,-41.737,179.004,5.784,149.325
C02398=1170.638,-96.815,-41.727,179.001,5.784,149.325
C02399=1170.643,-97.066,-41.717,179.000,5.784,149.326
C02400=1170.648,-97.315,-41.708,178.997,5.784,149.327
C02401=1170.654,-97.566,-41.698,178.995,5.783,149.327
C02402=1170.658,-97.815,-41.689,178.993,5.783,149.328
C02403=1170.664,-98.065,-41.679,178.991,5.782,149.328
C02404=1170.669,-98.314,-41.670,178.988,5.783,149.329
C02405=1170.675,-98.564,-41.660,178.986,5.782,149.329
C02406=1170.680,-98.814,-41.650,178.985,5.782,149.330
C02407=1170.686,-99.064,-41.641,178.982,5.782,149.331
C02408=1170.691,-99.313,-41.631,178.980,5.781,149.331
C02409=1170.696,-99.564,-41.621,178.978,5.781,149.332
C02410=1170.701,-99.813,-41.612,178.976,5.781,149.332
C02411=1170.707,-100.063,-41.602,178.973,5.781,149.333
C02412=1170.712,-100.312,-41.593,178.971,5.780,149.333
C02413=1170.718,-100.563,-41.583,178.969,5.779,149.334
C02414=1170.722,-100.812,-41.574,178.967,5.780,149.335
C02415=1170.728,-101.062,-41.564,178.965,5.779,149.335
C02416=1170.734,-101.312,-41.555,178.963,5.780,149.336
C02417=1170.738,-101.561,-41.546,178.961,5.779,149.336
C02418=1170.745,-101.833,-41.535,178.958,5.778,149.337
C02419=1170.750,-102.105,-41.525,178.956,5.778,149.338
C02420=1170.756,-102.377,-41.514,178.954,5.778,149.338
C02421=1170.762,-102.648,-41.504,178.951,5.778,149.339
C02422=1170.768,-102.899,-41.495,178.949,5.778,149.339
C02423=1170.772,-103.148,-41.485,178.947,5.777,149.340
C02424=1170.778,-103.399,-41.476,178.945,5.777,149.341
C02425=1170.783,-103.648,-41.466,178.943,5.777,149.341
C02426=1170.788,-103.898,-41.457,178.941,5.777,149.342
C02427=1170.794,-104.148,-41.448,178.939,5.776,149.342
C02428=1170.799,-104.397,-41.438,178.936,5.776,149.343
C02429=1170.804,-104.647,-41.429,178.934,5.776,149.344
C02430=1170.810,-104.897,-41.419,178.932,5.775,149.344
C02431=1170.815,-105.146,-41.410,178.930,5.775,149.345
C02432=1170.820,-105.396,-41.401,178.928,5.775,149.345
C02433=1170.826,-105.646,-41.391,178.926,5.775,149.346
C02434=1170.830,-105.896,-41.382,178.924,5.774,149.346
C02435=1170.836,-106.146,-41.372,178.921,5.774,149.347
C02436=1170.842,-106.396,-41.363,178.919,5.774,149.348
C02437=1170.846,-106.645,-41.354,178.917,5.773,149.348
C02438=1170.852,-106.895,-41.344,178.915,5.774,149.349
C02439=1170.857,-107.145,-41.335,178.913,5.773,149.349
C02440=1170.862,-107.394,-41.326,178.911,5.773,149.350
C02441=1170.867,-107.644,-41.317,178.909,5.772,149.351
C02442=1170.873,-107.894,-41.307,178.907,5.772,149.351
C02443=1170.879,-108.144,-41.299,178.904,5.772,149.352
C02444=1170.883,-108.393,-41.289,178.903,5.772,149.352
C02445=1170.889,-108.643,-41.279,178.900,5.772,149.353
C02446=1170.894,-108.893,-41.271,178.898,5.771,149.353
C02447=1170.900,-109.143,-41.262,178.896,5.771,149.354
C02448=1170.905,-109.393,-41.251,178.894,5.771,149.355
C02449=1170.910,-109.642,-41.243,178.892,5.771,149.355
C02450=1170.916,-109.892,-41.234,178.889,5.770,149.356
C02451=1170.921,-110.141,-41.225,178.888,5.770,149.356
C02452=1170.927,-110.392,-41.216,178.885,5.770,149.357
C02453=1170.932,-110.641,-41.206,178.883,5.770,149.357
C02454=1170.937,-110.891,-41.197,178.881,5.769,149.358
C02455=1170.942,-111.141,-41.188,178.879,5.770,149.359
C02456=1170.948,-111.391,-41.179,178.877,5.769,149.359
C02457=1170.954,-111.641,-41.170,178.875,5.769,149.360
C02458=1170.959,-111.890,-41.161,178.873,5.768,149.360
C02459=1170.964,-112.140,-41.151,178.870,5.768,149.361
C02460=1170.969,-112.390,-41.142,178.868,5.768,149.362
C02461=1170.975,-112.640,-41.133,178.866,5.767,149.362
C02462=1170.980,-112.890,-41.124,178.865,5.767,149.363
C02463=1170.985,-113.139,-41.115,178.862,5.767,149.363
C02464=1170.991,-113.390,-41.106,178.860,5.767,149.364
C02465=1170.997,-113.639,-41.097,178.858,5.766,149.364
C02466=1171.001,-113.888,-41.088,178.856,5.767,149.365
C02467=1171.007,-114.138,-41.079,178.854,5.766,149.365
C02468=1171.012,-114.388,-41.070,178.852,5.766,149.366
C02469=1171.018,-114.638,-41.060,178.850,5.766,149.367
C02470=1171.023,-114.888,-41.051,178.848,5.766,149.367
C02471=1171.028,-115.138,-41.042,178.845,5.765,149.368
C02472=1171.033,-115.387,-41.034,178.844,5.765,149.368
C02473=1171.038,-115.637,-41.025,178.841,5.764,149.369
C02474=1171.044,-115.886,-41.016,178.839,5.765,149.370
C02475=1171.050,-116.137,-41.007,178.837,5.764,149.370
C02476=1171.055,-116.386,-40.998,178.836,5.764,149.370
C02477=1171.060,-116.636,-40.989,178.833,5.764,149.371
C02478=1171.066,-116.886,-40.980,178.831,5.763,149.372
C02479=1171.071,-117.136,-40.971,178.829,5.763,149.372
C02480=1171.076,-117.386,-40.962,178.826,5.763,149.373
C02481=1171.081,-117.636,-40.953,178.825,5.763,149.373
C02482=1171.088,-117.885,-40.944,178.822,5.762,149.374
C02483=1171.093,-118.135,-40.935,178.821,5.762,149.375
C02484=1171.098,-118.385,-40.926,178.818,5.762,149.375
C02485=1171.103,-118.635,-40.917,178.816,5.762,149.376
C02486=1171.108,-118.884,-40.908,178.814,5.761,149.376
C02487=1171.113,-119.134,-40.900,178.813,5.761,149.377
C02488=1171.119,-119.383,-40.891,178.810,5.761,149.377
C02489=1171.124,-119.633,-40.882,178.808,5.761,149.378
C02490=1171.129,-119.883,-40.873,178.806,5.760,149.378
C02491=1171.135,-120.133,-40.864,178.804,5.761,149.379
C02492=1171.141,-120.383,-40.855,178.802,5.760,149.380
C02493=1171.146,-120.633,-40.846,178.800,5.760,149.380
C02494=1171.151,-120.882,-40.837,178.797,5.759,149.381
C02495=1171.157,-121.132,-40.829,178.796,5.759,149.381
C02496=1171.162,-121.382,-40.820,178.794,5.759,149.382
C02497=1171.167,-121.632,-40.811,178.792,5.759,149.383
C02498=1171.172,-121.882,-40.802,178.789,5.758,149.383
C02499=1171.178,-122.131,-40.793,178.787,5.759,149.384
C02500=1171.183,-122.381,-40.785,178.785,5.758,149.384
C02501=1171.189,-122.631,-40.776,178.784,5.758,149.385
C02502=1171.194,-122.881,-40.767,178.781,5.757,149.385
C02503=1171.199,-123.131,-40.758,178.779,5.758,149.386
C02504=1171.205,-123.380,-40.750,178.777,5.757,149.386
C02505=1171.210,-123.630,-40.741,178.775,5.757,149.387
C02506=1171.215,-123.880,-40.732,178.773,5.757,149.388
C02507=1171.220,-124.129,-40.723,178.771,5.757,149.388
C02508=1171.226,-124.380,-40.715,178.769,5.756,149.389
C02509=1171.231,-124.629,-40.707,178.767,5.756,149.389
C02510=1171.237,-124.879,-40.698,178.765,5.756,149.390
C02511=1171.242,-125.129,-40.689,178.763,5.756,149.390
C02512=1171.247,-125.379,-40.680,178.760,5.755,149.391
C02513=1171.253,-125.628,-40.671,178.759,5.755,149.391
C02514=1171.258,-125.878,-40.663,178.757,5.754,149.392
C02515=1171.263,-126.128,-40.654,178.755,5.755,149.393
C02516=1171.268,-126.378,-40.645,178.752,5.754,149.393
C02517=1171.274,-126.627,-40.637,178.751,5.754,149.394
C02518=1171.279,-126.877,-40.628,178.748,5.754,149.394
C02519=1171.285,-127.127,-40.620,178.746,5.754,149.395
C02520=1171.290,-127.377,-40.611,178.744,5.753,149.395
C02521=1171.296,-127.626,-40.602,178.742,5.754,149.396
C02522=1170.875,-127.638,-40.643,178.739,5.756,149.398
C02523=1170.869,-127.389,-40.652,178.741,5.757,149.397
C02524=1170.864,-127.138,-40.660,178.743,5.757,149.397
C02525=1170.859,-126.888,-40.669,178.745,5.758,149.396
C02526=1170.853,-126.639,-40.678,178.747,5.757,149.395
C02527=1170.848,-126.389,-40.686,178.749,5.758,149.395
C02528=1170.842,-126.139,-40.695,178.751,5.758,149.395
C02529=1170.837,-125.889,-40.704,178.753,5.759,149.394
C02530=1170.831,-125.640,-40.712,178.755,5.758,149.393
C02531=1170.826,-125.390,-40.721,178.757,5.759,149.393
C02532=1170.821,-125.140,-40.730,178.759,5.759,149.392
C02533=1170.815,-124.890,-40.738,178.761,5.760,149.392
C02534=1170.810,-124.640,-40.747,178.763,5.760,149.391
C02535=1170.805,-124.391,-40.755,178.766,5.760,149.390
C02536=1170.799,-124.141,-40.764,178.767,5.760,149.390
C02537=1170.794,-123.891,-40.773,178.770,5.761,149.389
C02538=1170.789,-123.641,-40.782,178.771,5.761,149.389
C02539=1170.783,-123.392,-40.791,178.774,5.761,149.388
C02540=1170.778,-123.141,-40.799,178.775,5.761,149.388
C02541=1170.773,-122.892,-40.808,178.778,5.762,149.387
C02542=1170.767,-122.642,-40.817,178.780,5.761,149.387
C02543=1170.762,-122.393,-40.825,178.782,5.762,149.386
C02544=1170.757,-122.143,-40.834,178.783,5.762,149.386
C02545=1170.751,-121.893,-40.843,178.786,5.762,149.385
C02546=1170.746,-121.643,-40.852,178.788,5.762,149.384
C02547=1170.741,-121.393,-40.861,178.790,5.763,149.384
C02548=1170.736,-121.143,-40.870,178.792,5.763,149.383
C02549=1170.730,-120.893,-40.878,178.794,5.763,149.383
C02550=1170.724,-120.643,-40.887,178.796,5.763,149.382
C02551=1170.719,-120.393,-40.896,178.798,5.764,149.381
C02552=1170.714,-120.144,-40.905,178.800,5.764,149.381
C02553=1170.708,-119.894,-40.914,178.802,5.765,149.381
C02554=1170.703,-119.645,-40.922,178.804,5.764,149.380
C02555=1170.697,-119.395,-40.931,178.807,5.765,149.379
C02556=1170.692,-119.145,-40.940,178.808,5.765,149.379
C02557=1170.687,-118.895,-40.949,178.811,5.765,149.378
C02558=1170.682,-118.645,-40.958,178.812,5.765,149.378
C02559=1170.677,-118.395,-40.967,178.815,5.766,149.377
C02560=1170.671,-118.146,-40.975,178.817,5.766,149.376
C02561=1170.665,-117.896,-40.985,178.819,5.766,149.376
C02562=1170.660,-117.646,-40.994,178.821,5.766,149.375
C02563=1170.655,-117.396,-41.003,178.823,5.767,149.375
C02564=1170.650,-117.146,-41.011,178.825,5.767,149.374
C02565=1170.644,-116.897,-41.020,178.827,5.767,149.374
C02566=1170.639,-116.647,-41.029,178.829,5.767,149.373
C02567=1170.633,-116.398,-41.038,178.831,5.768,149.373
C02568=1170.628,-116.148,-41.047,178.833,5.767,149.372
C02569=1170.622,-115.898,-41.056,178.836,5.768,149.371
C02570=1170.617,-115.648,-41.065,178.837,5.768,149.371
C02571=1170.612,-115.398,-41.074,178.840,5.768,149.370
C02572=1170.607,-115.148,-41.083,178.841,5.768,149.370
C02573=1170.602,-114.898,-41.092,178.844,5.769,149.369
C02574=1170.596,-114.649,-41.102,178.846,5.769,149.368
C02575=1170.591,-114.399,-41.111,178.848,5.770,149.368
C02576=1170.585,-114.150,-41.119,178.850,5.769,149.367
C02577=1170.580,-113.900,-41.128,178.852,5.770,149.367
C02578=1170.575,-113.650,-41.137,178.854,5.771,149.366
C02579=1170.570,-113.400,-41.146,178.856,5.770,149.366
C02580=1170.564,-113.150,-41.156,178.859,5.771,149.365
C02581=1170.559,-112.900,-41.164,178.861,5.771,149.364
C02582=1170.553,-112.650,-41.173,178.863,5.771,149.364
C02583=1170.549,-112.401,-41.183,178.864,5.771,149.363
C02584=1170.543,-112.151,-41.192,178.867,5.772,149.363
C02585=1170.538,-111.901,-41.201,178.869,5.772,149.362
C02586=1170.532,-111.651,-41.210,178.871,5.772,149.362
C02587=1170.527,-111.402,-41.219,178.873,5.772,149.361
C02588=1170.521,-111.152,-41.228,178.875,5.773,149.361
C02589=1170.516,-110.903,-41.238,178.877,5.772,149.360
C02590=1170.511,-110.653,-41.247,178.879,5.773,149.359
C02591=1170.506,-110.403,-41.256,178.881,5.773,149.359
C02592=1170.500,-110.153,-41.265,178.884,5.774,149.358
C02593=1170.494,-109.903,-41.274,178.886,5.774,149.358
C02594=1170.490,-109.654,-41.284,178.888,5.774,149.357
C02595=1170.484,-109.404,-41.293,178.890,5.775,149.356
C02596=1170.479,-109.154,-41.302,178.892,5.775,149.356
C02597=1170.473,-108.904,-41.311,178.895,5.775,149.355
C02598=1170.468,-108.654,-41.320,178.896,5.775,149.355
C02599=1170.463,-108.404,-41.330,178.898,5.776,149.354
C02600=1170.457,-108.155,-41.339,178.900,5.775,149.354
C02601=1170.452,-107.905,-41.348,178.903,5.776,149.353
C02602=1170.447,-107.655,-41.357,178.905,5.776,149.352
C02603=1170.441,-107.405,-41.367,178.907,5.776,149.352
C02604=1170.436,-107.155,-41.376,178.909,5.777,149.351
C02605=1170.431,-106.906,-41.385,178.911,5.777,149.351
C02606=1170.426,-106.656,-41.395,178.913,5.778,149.350
C02607=1170.420,-106.406,-41.404,178.915,5.777,149.349
C02608=1170.415,-106.156,-41.413,178.918,5.778,149.349
C02609=1170.409,-105.906,-41.422,178.919,5.778,149.349
C02610=1170.404,-105.657,-41.432,178.922,5.778,149.348
C02611=1170.399,-105.407,-41.441,178.923,5.778,149.347
C02612=1170.393,-105.157,-41.450,178.926,5.779,149.347
C02613=1170.389,-104.908,-41.460,178.928,5.779,149.346
C02614=1170.383,-104.658,-41.469,178.930,5.779,149.345
C02615=1170.377,-104.408,-41.478,178.933,5.780,149.345
C02616=1170.373,-104.158,-41.488,178.934,5.780,149.344
C02617=1170.367,-103.908,-41.497,178.937,5.780,149.344
C02618=1170.362,-103.659,-41.507,178.938,5.780,149.343
C02619=1170.357,-103.409,-41.516,178.941,5.780,149.343
C02620=1170.351,-103.159,-41.525,178.943,5.781,149.342
C02621=1170.346,-102.910,-41.535,178.945,5.781,149.342
C02622=1170.340,-102.660,-41.545,178.948,5.782,149.341
C02623=1170.335,-102.388,-41.555,178.949,5.782,149.340
C02624=1170.329,-102.116,-41.565,178.952,5.782,149.340
C02625=1170.324,-101.844,-41.575,178.955,5.782,149.339
C02626=1170.317,-101.573,-41.585,178.956,5.782,149.338
C02627=1170.312,-101.323,-41.595,178.959,5.783,149.338
C02628=1170.307,-101.073,-41.604,178.961,5.784,149.337
C02629=1170.301,-100.822,-41.614,178.963,5.783,149.337
C02630=1170.297,-100.573,-41.624,178.965,5.784,149.336
C02631=1170.291,-100.323,-41.633,178.967,5.783,149.335
C02632=1170.286,-100.074,-41.643,178.970,5.784,149.335
C02633=1170.281,-99.824,-41.652,178.972,5.785,149.334
C02634=1170.275,-99.574,-41.662,178.974,5.785,149.334
C02635=1170.270,-99.325,-41.671,178.976,5.785,149.333
C02636=1170.264,-99.075,-41.681,178.978,5.785,149.332
C02637=1170.259,-98.825,-41.690,178.980,5.786,149.332
C02638=1170.253,-98.576,-41.700,178.982,5.785,149.331
C02639=1170.248,-98.326,-41.709,178.985,5.786,149.331
C02640=1170.243,-98.076,-41.719,178.987,5.787,149.330
C02641=1170.238,-97.826,-41.728,178.989,5.786,149.330
C02642=1170.233,-97.576,-41.739,178.991,5.787,149.329
C02643=1170.227,-97.326,-41.748,178.993,5.787,149.328
C02644=1170.222,-97.077,-41.758,178.995,5.788,149.328
C02645=1170.217,-96.827,-41.767,178.998,5.788,149.327
C02646=1170.211,-96.577,-41.777,179.000,5.788,149.327
C02647=1170.206,-96.328,-41.786,179.002,5.788,149.326
C02648=1170.200,-96.078,-41.796,179.004,5.788,149.325
C02649=1170.195,-95.828,-41.807,179.006,5.789,149.325
C02650=1170.190,-95.578,-41.815,179.008,5.789,149.324
C02651=1170.184,-95.328,-41.826,179.010,5.789,149.324
C02652=1170.179,-95.078,-41.835,179.013,5.790,149.323
C02653=1170.174,-94.829,-41.845,179.015,5.790,149.323
C02654=1170.169,-94.580,-41.854,179.017,5.790,149.322
C02655=1170.163,-94.330,-41.864,179.019,5.790,149.321
C02656=1170.159,-94.080,-41.874,179.022,5.791,149.321
C02657=1170.153,-93.830,-41.884,179.024,5.791,149.320
C02658=1170.147,-93.580,-41.894,179.026,5.791,149.320
C02659=1170.142,-93.331,-41.903,179.028,5.792,149.319
C02660=1170.136,-93.080,-41.913,179.030,5.792,149.319
C02661=1170.132,-92.831,-41.922,179.032,5.792,149.318
C02662=1170.127,-92.581,-41.933,179.034,5.793,149.317
C02663=1170.121,-92.331,-41.942,179.037,5.792,149.317
C02664=1170.116,-92.082,-41.952,179.039,5.793,149.316
C02665=1170.110,-91.832,-41.962,179.041,5.794,149.315
C02666=1170.105,-91.582,-41.971,179.043,5.794,149.315
C02667=1170.099,-91.333,-41.981,179.046,5.794,149.314
C02668=1170.094,-91.082,-41.992,179.047,5.794,149.314
C02669=1170.090,-90.833,-42.001,179.050,5.794,149.313
C02670=1170.084,-90.583,-42.011,179.052,5.795,149.313
C02671=1170.078,-90.334,-42.021,179.054,5.795,149.312
C02672=1170.074,-90.084,-42.031,179.056,5.796,149.311
C02673=1170.068,-89.833,-42.041,179.058,5.795,149.311
C02674=1170.062,-89.584,-42.051,179.061,5.796,149.310
C02675=1170.057,-89.335,-42.060,179.063,5.797,149.310
C02676=1170.052,-89.085,-42.071,179.065,5.796,149.309
C02677=1170.047,-88.835,-42.081,179.067,5.797,149.309
C02678=1170.042,-88.585,-42.090,179.070,5.797,149.308
C02679=1170.036,-88.335,-42.100,179.071,5.797,149.307
C02680=1170.030,-88.086,-42.111,179.074,5.798,149.307
C02681=1170.026,-87.836,-42.121,179.076,5.798,149.306
C02682=1170.020,-87.586,-42.130,179.078,5.798,149.305
C02683=1170.015,-87.336,-42.140,179.081,5.799,149.305
C02684=1170.010,-87.087,-42.150,179.083,5.799,149.304
C02685=1170.005,-86.837,-42.160,179.085,5.799,149.304
C02686=1169.999,-86.587,-42.171,179.088,5.800,149.303
C02687=1169.994,-86.338,-42.180,179.089,5.800,149.303
C02688=1169.988,-86.088,-42.190,179.092,5.800,149.302
C02689=1169.983,-85.838,-42.200,179.093,5.800,149.301
C02690=1169.978,-85.588,-42.211,179.096,5.801,149.301
C02691=1169.973,-85.339,-42.220,179.098,5.801,149.300
C02692=1169.967,-85.089,-42.230,179.100,5.801,149.299
C02693=1169.962,-84.839,-42.241,179.102,5.802,149.299
C02694=1169.957,-84.590,-42.251,179.105,5.802,149.298
C02695=1169.952,-84.340,-42.260,179.107,5.802,149.298
C02696=1169.947,-84.089,-42.271,179.109,5.802,149.297
C02697=1169.941,-83.840,-42.281,179.112,5.803,149.297
C02698=1169.935,-83.590,-42.291,179.114,5.803,149.296
C02699=1169.931,-83.340,-42.301,179.116,5.804,149.295
C02700=1169.926,-83.091,-42.311,179.118,5.803,149.295
C02701=1169.920,-82.841,-42.321,179.120,5.804,149.294
C02702=1169.914,-82.592,-42.332,179.123,5.804,149.293
C02703=1169.909,-82.342,-42.342,179.124,5.804,149.293
C02704=1169.905,-82.092,-42.352,179.127,5.805,149.292
C02705=1169.899,-81.843,-42.362,179.129,5.806,149.292
C02706=1169.894,-81.592,-42.373,179.131,5.805,149.291
C02707=1169.888,-81.343,-42.383,179.134,5.806,149.291
C02708=1169.883,-81.093,-42.393,179.136,5.806,149.290
C02709=1169.878,-80.843,-42.404,179.138,5.806,149.289
C02710=1169.873,-80.594,-42.413,179.140,5.807,149.289
C02711=1169.867,-80.344,-42.423,179.143,5.808,149.288
C02712=1169.862,-80.094,-42.434,179.145,5.807,149.288
C02713=1169.857,-79.845,-42.444,179.147,5.808,149.287
C02714=1169.851,-79.595,-42.454,179.150,5.808,149.286
C02715=1169.846,-79.345,-42.465,179.151,5.808,149.286
C02716=1169.841,-79.095,-42.475,179.154,5.809,149.285
C02717=1169.836,-78.845,-42.485,179.156,5.809,149.285
C02718=1169.831,-78.596,-42.495,179.158,5.809,149.284
C02719=1169.825,-78.346,-42.506,179.160,5.810,149.283
C02720=1169.820,-78.096,-42.516,179.163,5.810,149.283
C02721=1169.814,-77.846,-42.526,179.165,5.810,149.282
C02722=1169.809,-77.597,-42.537,179.167,5.811,149.282
C02723=1169.804,-77.347,-42.547,179.169,5.811,149.281
C02724=1169.798,-77.097,-42.557,179.172,5.811,149.280
C02725=1169.793,-76.847,-42.568,179.174,5.812,149.280
C02726=1169.788,-76.597,-42.578,179.176,5.812,149.279
C02727=1169.783,-76.327,-42.590,179.178,5.812,149.279
C02728=1169.776,-76.056,-42.601,179.181,5.813,149.278
C02729=1169.771,-75.784,-42.612,179.183,5.813,149.277
C02730=1169.765,-75.513,-42.623,179.186,5.813,149.277
C02731=1169.760,-75.263,-42.634,179.188,5.814,149.276
C02732=1169.754,-75.014,-42.645,179.190,5.814,149.275
C02733=1169.749,-74.764,-42.655,179.192,5.815,149.275
C02734=1169.744,-74.515,-42.665,179.195,5.815,149.274
C02735=1169.739,-74.264,-42.676,179.197,5.815,149.274
C02736=1169.733,-74.015,-42.686,179.199,5.815,149.273
C02737=1169.727,-73.765,-42.696,179.202,5.816,149.273
C02738=1169.723,-73.516,-42.708,179.204,5.816,149.272
C02739=1169.717,-73.266,-42.718,179.206,5.817,149.271
C02740=1169.712,-73.016,-42.728,179.209,5.817,149.271
C02741=1169.707,-72.766,-42.739,179.210,5.817,149.270
C02742=1169.702,-72.516,-42.749,179.213,5.817,149.269
C02743=1169.696,-72.267,-42.760,179.215,5.818,149.269
C02744=1169.691,-72.017,-42.771,179.217,5.818,149.268
C02745=1169.686,-71.767,-42.781,179.220,5.818,149.268
C02746=1169.680,-71.518,-42.791,179.222,5.819,149.267
C02747=1169.675,-71.268,-42.802,179.224,5.819,149.266
C02748=1169.670,-71.019,-42.813,179.226,5.819,149.266
C02749=1169.665,-70.768,-42.823,179.229,5.820,149.265
C02750=1169.659,-70.519,-42.833,179.231,5.821,149.265
C02751=1169.655,-70.269,-42.845,179.233,5.820,149.264
C02752=1169.649,-70.020,-42.855,179.235,5.821,149.264
C02753=1169.644,-69.769,-42.865,179.238,5.821,149.263
C02754=1169.639,-69.521,-42.876,179.240,5.821,149.262
C02755=1169.634,-69.270,-42.887,179.242,5.822,149.262
C02756=1169.628,-69.021,-42.897,179.244,5.823,149.261
C02757=1169.623,-68.770,-42.908,179.247,5.822,149.260
C02758=1169.618,-68.522,-42.919,179.249,5.823,149.260
C02759=1169.613,-68.271,-42.929,179.251,5.823,149.259
C02760=1169.607,-68.022,-42.941,179.254,5.824,149.259
C02761=1169.602,-67.772,-42.951,179.256,5.824,149.258
C02762=1169.596,-67.522,-42.962,179.258,5.824,149.257
C02763=1169.591,-67.273,-42.973,179.261,5.825,149.257
C02764=1169.586,-67.023,-42.983,179.263,5.825,149.256
C02765=1169.581,-66.773,-42.994,179.265,5.825,149.256
C02766=1169.576,-66.524,-43.005,179.267,5.826,149.255
C02767=1169.571,-66.274,-43.015,179.270,5.827,149.254
C02768=1169.565,-66.025,-43.026,179.272,5.826,149.254
C02769=1169.560,-65.774,-43.037,179.274,5.827,149.253
C02770=1169.555,-65.524,-43.048,179.277,5.827,149.253
C02771=1169.549,-65.275,-43.059,179.279,5.827,149.252
C02772=1169.544,-65.025,-43.069,179.281,5.828,149.251
C02773=1169.539,-64.776,-43.080,179.283,5.828,149.251
C02774=1169.534,-64.526,-43.091,179.286,5.829,149.250
C02775=1169.528,-64.276,-43.102,179.288,5.829,149.250
C02776=1169.523,-64.026,-43.113,179.290,5.829,149.249
C02777=1169.518,-63.777,-43.124,179.293,5.830,149.248
C02778=1169.513,-63.527,-43.134,179.295,5.831,149.248
C02779=1169.508,-63.277,-43.145,179.297,5.830,149.247
C02780=1169.502,-63.028,-43.156,179.299,5.831,149.247
C02781=1169.497,-62.777,-43.167,179.302,5.831,149.246
C02782=1169.491,-62.528,-43.178,179.304,5.831,149.245
C02783=1169.486,-62.278,-43.189,179.306,5.832,149.245
C02784=1169.482,-62.028,-43.200,179.309,5.832,149.244
C02785=1169.476,-61.779,-43.211,179.311,5.833,149.244
C02786=1169.471,-61.529,-43.222,179.313,5.833,149.243
C02787=1169.465,-61.280,-43.233,179.315,5.833,149.242
C02788=1169.460,-61.030,-43.243,179.318,5.834,149.242
C02789=1169.456,-60.780,-43.255,179.320,5.835,149.241
C02790=1169.449,-60.530,-43.266,179.322,5.834,149.241
C02791=1169.445,-60.281,-43.277,179.325,5.835,149.240
C02792=1169.439,-60.031,-43.287,179.327,5.835,149.239
C02793=1169.434,-59.782,-43.298,179.330,5.836,149.239
C02794=1169.429,-59.532,-43.310,179.331,5.836,149.238
C02795=1169.423,-59.282,-43.320,179.334,5.836,149.237
C02796=1169.419,-59.032,-43.332,179.336,5.837,149.237
C02797=1169.413,-58.782,-43.343,179.339,5.837,149.236
C02798=1169.408,-58.533,-43.354,179.341,5.837,149.236
C02799=1169.403,-58.283,-43.365,179.343,5.838,149.235
C02800=1169.398,-58.033,-43.376,179.346,5.838,149.234
C02801=1169.392,-57.784,-43.387,179.348,5.839,149.234
C02802=1169.387,-57.534,-43.398,179.350,5.839,149.233
C02803=1169.382,-57.284,-43.409,179.352,5.839,149.233
C02804=1169.376,-57.035,-43.421,179.355,5.840,149.232
C02805=1169.371,-56.785,-43.432,179.357,5.841,149.232
C02806=1169.366,-56.535,-43.442,179.359,5.840,149.231
C02807=1169.360,-56.286,-43.454,179.362,5.841,149.230
C02808=1169.356,-56.036,-43.465,179.364,5.842,149.230
C02809=1169.351,-55.786,-43.476,179.367,5.842,149.229
C02810=1169.345,-55.537,-43.487,179.368,5.842,149.228
C02811=1169.340,-55.287,-43.499,179.371,5.842,149.228
C02812=1169.335,-55.037,-43.510,179.373,5.843,149.227
C02813=1169.330,-54.787,-43.521,179.376,5.844,149.227
C02814=1169.324,-54.538,-43.532,179.378,5.843,149.226
C02815=1169.320,-54.288,-43.543,179.380,5.844,149.225
C02816=1169.314,-54.038,-43.555,179.383,5.844,149.225
C02817=1169.309,-53.789,-43.565,179.385,5.845,149.224
C02818=1169.304,-53.539,-43.577,179.387,5.846,149.224
C02819=1169.298,-53.289,-43.589,179.389,5.846,149.223
C02820=1169.294,-53.040,-43.600,179.392,5.846,149.222
C02821=1169.287,-52.790,-43.611,179.394,5.846,149.222
C02822=1169.283,-52.540,-43.622,179.397,5.847,149.221
C02823=1169.277,-52.290,-43.634,179.399,5.847,149.220
C02824=1169.272,-52.041,-43.645,179.401,5.848,149.220
C02825=1169.267,-51.792,-43.656,179.403,5.848,149.219
C02826=1169.262,-51.542,-43.668,179.406,5.849,149.219
C02827=1169.257,-51.291,-43.679,179.408,5.849,149.218
C02828=1169.251,-51.042,-43.690,179.410,5.849,149.217
C02829=1169.246,-50.793,-43.701,179.413,5.850,149.217
C02830=1169.241,-50.543,-43.713,179.415,5.850,149.216
C02831=1169.235,-50.272,-43.725,179.418,5.851,149.216
C02832=1169.230,-50.002,-43.737,179.420,5.851,149.215
C02833=1169.224,-49.731,-43.750,179.423,5.852,149.214
C02834=1169.218,-49.462,-43.762,179.425,5.852,149.214
C02835=1169.213,-49.211,-43.773,179.428,5.853,149.213
C02836=1169.208,-48.961,-43.785,179.430,5.853,149.212
C02837=1169.203,-48.712,-43.797,179.432,5.853,149.212
C02838=1169.198,-48.462,-43.808,179.435,5.854,149.211
C02839=1169.192,-48.213,-43.819,179.437,5.854,149.211
C02840=1169.187,-47.963,-43.831,179.439,5.854,149.210
C02841=1169.182,-47.713,-43.843,179.441,5.855,149.209
C02842=1169.177,-47.463,-43.854,179.444,5.855,149.209
C02843=1169.172,-47.214,-43.866,179.446,5.856,149.208
C02844=1169.166,-46.965,-43.877,179.449,5.856,149.208
C02845=1169.161,-46.715,-43.889,179.451,5.857,149.207
C02846=1169.155,-46.465,-43.901,179.453,5.857,149.206
C02847=1169.151,-46.215,-43.912,179.455,5.858,149.206
C02848=1169.145,-45.965,-43.924,179.458,5.858,149.205
C02849=1169.140,-45.716,-43.935,179.461,5.858,149.204
C02850=1169.135,-45.466,-43.946,179.463,5.859,149.204
C02851=1169.130,-45.217,-43.958,179.465,5.859,149.203
C02852=1169.124,-44.967,-43.970,179.467,5.860,149.203
C02853=1169.119,-44.717,-43.982,179.470,5.860,149.202
C02854=1169.114,-44.467,-43.993,179.472,5.860,149.201
C02855=1169.109,-44.217,-44.005,179.475,5.861,149.201
C02856=1169.104,-43.968,-44.016,179.477,5.861,149.200
C02857=1169.098,-43.718,-44.028,179.479,5.862,149.200
C02858=1169.093,-43.468,-44.039,179.482,5.862,149.199
C02859=1169.088,-43.219,-44.051,179.484,5.863,149.199
C02860=1169.083,-42.969,-44.063,179.486,5.863,149.198
C02861=1169.078,-42.719,-44.074,179.489,5.864,149.197
C02862=1169.073,-42.470,-44.086,179.491,5.864,149.197
C02863=1169.067,-42.221,-44.098,179.493,5.864,149.196
C02864=1169.062,-41.971,-44.109,179.496,5.865,149.196
C02865=1169.057,-41.721,-44.121,179.498,5.865,149.195
C02866=1169.051,-41.471,-44.133,179.501,5.866,149.194
C02867=1169.047,-41.222,-44.144,179.503,5.867,149.194
C02868=1169.041,-40.972,-44.156,179.505,5.866,149.193
C02869=1169.036,-40.722,-44.168,179.507,5.867,149.192
C02870=1169.031,-40.473,-44.180,179.510,5.867,149.192
C02871=1169.026,-40.223,-44.192,179.513,5.868,149.191
C02872=1169.020,-39.973,-44.204,179.515,5.869,149.191
C02873=1169.015,-39.724,-44.215,179.517,5.869,149.190
C02874=1169.010,-39.474,-44.227,179.519,5.869,149.189
C02875=1169.005,-39.225,-44.239,179.522,5.870,149.189
C02876=1168.999,-38.975,-44.251,179.524,5.870,149.188
C02877=1168.994,-38.725,-44.262,179.527,5.871,149.188
C02878=1168.989,-38.475,-44.274,179.529,5.871,149.187
C02879=1168.984,-38.225,-44.286,179.531,5.872,149.186
C02880=1168.979,-37.976,-44.298,179.534,5.872,149.186
C02881=1168.974,-37.726,-44.310,179.536,5.872,149.185
C02882=1168.968,-37.476,-44.322,179.538,5.873,149.185
C02883=1168.963,-37.226,-44.334,179.541,5.873,149.184
C02884=1168.959,-36.977,-44.346,179.543,5.874,149.183
C02885=1168.953,-36.727,-44.358,179.546,5.875,149.183
C02886=1168.948,-36.478,-44.370,179.548,5.875,149.182
C02887=1168.943,-36.228,-44.382,179.550,5.875,149.181
C02888=1168.937,-35.978,-44.394,179.553,5.875,149.181
C02889=1168.932,-35.729,-44.405,179.555,5.876,149.180
C02890=1168.926,-35.479,-44.417,179.558,5.877,149.180
C02891=1168.921,-35.230,-44.430,179.560,5.877,149.179
C02892=1168.916,-34.980,-44.441,179.562,5.878,149.178
C02893=1168.911,-34.731,-44.453,179.565,5.878,149.178
C02894=1168.906,-34.481,-44.465,179.567,5.878,149.177
C02895=1168.901,-34.231,-44.477,179.569,5.879,149.177
C02896=1168.895,-33.981,-44.489,179.572,5.880,149.176
C02897=1168.890,-33.732,-44.502,179.574,5.880,149.175
C02898=1168.885,-33.482,-44.514,179.577,5.880,149.175
C02899=1168.880,-33.233,-44.526,179.579,5.881,149.174
C02900=1168.875,-32.983,-44.538,179.582,5.882,149.174
C02901=1168.869,-32.733,-44.549,179.584,5.883,149.173
C02902=1168.864,-32.484,-44.562,179.586,5.882,149.172
C02903=1168.859,-32.234,-44.574,179.589,5.883,149.172
C02904=1168.854,-31.984,-44.587,179.591,5.883,149.171
C02905=1168.849,-31.734,-44.599,179.593,5.884,149.170
C02906=1168.845,-31.485,-44.611,179.596,5.885,149.170
C02907=1168.839,-31.235,-44.623,179.598,5.885,149.169
C02908=1168.834,-30.985,-44.635,179.601,5.886,149.169
C02909=1168.829,-30.736,-44.647,179.603,5.886,149.168
C02910=1168.823,-30.486,-44.659,179.606,5.887,149.167
C02911=1168.818,-30.237,-44.672,179.607,5.887,149.167
C02912=1168.813,-29.987,-44.683,179.610,5.887,149.166
C02913=1168.807,-29.737,-44.696,179.613,5.888,149.166
C02914=1168.802,-29.487,-44.708,179.615,5.888,149.165
C02915=1168.797,-29.238,-44.721,179.618,5.889,149.164
C02916=1168.792,-28.988,-44.732,179.620,5.890,149.164
C02917=1168.787,-28.739,-44.744,179.622,5.890,149.163
C02918=1168.782,-28.489,-44.756,179.625,5.891,149.163
C02919=1168.776,-28.240,-44.769,179.627,5.891,149.162
C02920=1168.772,-27.990,-44.782,179.629,5.891,149.161
C02921=1168.767,-27.740,-44.794,179.632,5.892,149.161
C02922=1168.761,-27.491,-44.806,179.634,5.892,149.160
C02923=1168.756,-27.241,-44.818,179.637,5.893,149.159
C02924=1168.751,-26.991,-44.831,179.639,5.894,149.159
C02925=1168.745,-26.741,-44.843,179.642,5.894,149.158
C02926=1168.740,-26.492,-44.855,179.644,5.894,149.158
C02927=1168.735,-26.243,-44.868,179.647,5.895,149.157
C02928=1168.730,-25.993,-44.880,179.649,5.896,149.156
C02929=1168.725,-25.743,-44.893,179.651,5.896,149.156
C02930=1168.720,-25.493,-44.905,179.653,5.896,149.155
C02931=1168.715,-25.244,-44.917,179.656,5.897,149.155
C02932=1168.710,-24.994,-44.930,179.658,5.897,149.154
C02933=1168.704,-24.744,-44.942,179.661,5.898,149.153
C02934=1168.699,-24.495,-44.954,179.663,5.899,149.153
C02935=1168.694,-24.225,-44.968,179.666,5.899,149.152
C02936=1168.688,-23.955,-44.982,179.668,5.899,149.152
C02937=1168.682,-23.686,-44.995,179.671,5.900,149.151
C02938=1168.677,-23.415,-45.008,179.674,5.900,149.150
C02939=1168.672,-23.166,-45.021,179.676,5.901,149.150
C02940=1168.666,-22.916,-45.034,179.679,5.902,149.149
C02941=1168.661,-22.667,-45.046,179.681,5.902,149.149
C02942=1168.656,-22.417,-45.058,179.683,5.903,149.148
C02943=1168.651,-22.167,-45.071,179.686,5.903,149.147
C02944=1168.646,-21.918,-45.084,179.688,5.904,149.147
C02945=1168.641,-21.668,-45.096,179.691,5.905,149.146
C02946=1168.635,-21.418,-45.108,179.693,5.905,149.146
C02947=1168.630,-21.169,-45.121,179.696,5.906,149.145
C02948=1168.626,-20.919,-45.134,179.698,5.906,149.144
C02949=1168.621,-20.670,-45.146,179.701,5.907,149.144
C02950=1168.614,-20.419,-45.159,179.703,5.907,149.143
C02951=1168.609,-20.170,-45.172,179.706,5.908,149.142
C02952=1168.604,-19.921,-45.184,179.708,5.909,149.142
C02953=1168.600,-19.671,-45.197,179.710,5.908,149.141
C02954=1168.594,-19.422,-45.210,179.712,5.909,149.141
C02955=1168.589,-19.172,-45.222,179.715,5.910,149.140
C02956=1168.584,-18.922,-45.234,179.718,5.910,149.139
C02957=1168.578,-18.673,-45.247,179.720,5.911,149.139
C02958=1168.574,-18.423,-45.260,179.723,5.911,149.138
C02959=1168.568,-18.173,-45.273,179.725,5.912,149.138
C02960=1168.563,-17.924,-45.286,179.727,5.913,149.137
C02961=1168.558,-17.675,-45.298,179.730,5.913,149.136
C02962=1168.553,-17.424,-45.311,179.732,5.914,149.136
C02963=1168.547,-17.174,-45.324,179.735,5.914,149.135
C02964=1168.542,-16.925,-45.336,179.737,5.915,149.135
C02965=1168.537,-16.676,-45.349,179.740,5.916,149.134
C02966=1168.533,-16.426,-45.362,179.742,5.916,149.133
C02967=1168.527,-16.176,-45.375,179.745,5.917,149.133
C02968=1168.522,-15.927,-45.388,179.747,5.917,149.132
C02969=1168.517,-15.677,-45.400,179.749,5.918,149.132
C02970=1168.512,-15.427,-45.413,179.752,5.919,149.131
C02971=1168.506,-15.178,-45.426,179.755,5.919,149.130
C02972=1168.501,-14.929,-45.439,179.757,5.920,149.130
C02973=1168.497,-14.679,-45.452,179.760,5.920,149.129
C02974=1168.491,-14.429,-45.464,179.762,5.921,149.129
C02975=1168.486,-14.180,-45.478,179.764,5.922,149.128
C02976=1168.481,-13.930,-45.491,179.766,5.921,149.127
C02977=1168.476,-13.680,-45.503,179.769,5.922,149.127
C02978=1168.471,-13.431,-45.516,179.771,5.922,149.126
C02979=1168.465,-13.181,-45.529,179.774,5.923,149.125
C02980=1168.460,-12.931,-45.542,179.776,5.924,149.125
C02981=1168.455,-12.682,-45.555,179.779,5.924,149.124
C02982=1168.449,-12.432,-45.568,179.781,5.925,149.124
C02983=1168.445,-12.182,-45.581,179.784,5.925,149.123
C02984=1168.440,-11.933,-45.593,179.786,5.926,149.122
C02985=1168.434,-11.683,-45.607,179.788,5.927,149.122
C02986=1168.429,-11.433,-45.620,179.791,5.927,149.121
C02987=1168.424,-11.184,-45.632,179.793,5.928,149.121
C02988=1168.419,-10.935,-45.645,179.796,5.928,149.120
C02989=1168.414,-10.684,-45.658,179.799,5.929,149.119
C02990=1168.409,-10.436,-45.672,179.801,5.930,149.119
C02991=1168.404,-10.185,-45.685,179.803,5.930,149.118
C02992=1168.399,-9.936,-45.698,179.806,5.931,149.118
C02993=1168.394,-9.687,-45.710,179.808,5.931,149.117
C02994=1168.388,-9.436,-45.724,179.811,5.932,149.116
C02995=1168.383,-9.187,-45.737,179.813,5.933,149.116
C02996=1168.378,-8.938,-45.749,179.816,5.933,149.115
C02997=1168.373,-8.688,-45.763,179.818,5.934,149.115
C02998=1168.368,-8.439,-45.776,179.821,5.934,149.114
C02999=1168.363,-8.188,-45.790,179.823,5.935,149.113
C03000=1168.358,-7.939,-45.802,179.825,5.936,149.113
C03001=1168.352,-7.690,-45.815,179.828,5.936,149.112
C03002=1168.348,-7.440,-45.829,179.830,5.937,149.112
C03003=1168.342,-7.191,-45.842,179.833,5.937,149.111
C03004=1168.337,-6.940,-45.855,179.836,5.938,149.110
C03005=1168.332,-6.691,-45.868,179.838,5.939,149.110
C03006=1168.326,-6.441,-45.881,179.840,5.939,149.109
C03007=1168.322,-6.192,-45.895,179.843,5.940,149.109
C03008=1168.317,-5.943,-45.907,179.845,5.940,149.108
C03009=1168.312,-5.692,-45.921,179.848,5.941,149.107
C03010=1168.307,-5.444,-45.934,179.850,5.942,149.107
C03011=1168.301,-5.193,-45.948,179.853,5.942,149.106
C03012=1168.296,-4.944,-45.960,179.855,5.943,149.105
C03013=1168.290,-4.694,-45.974,179.857,5.943,149.105
C03014=1168.286,-4.445,-45.987,179.860,5.944,149.104
C03015=1168.280,-4.195,-46.000,179.862,5.945,149.104
C03016=1168.276,-3.945,-46.013,179.865,5.945,149.103
C03017=1168.270,-3.696,-46.027,179.868,5.946,149.102
C03018=1168.266,-3.446,-46.040,179.870,5.947,149.102
C03019=1168.260,-3.197,-46.053,179.873,5.948,149.101
C03020=1168.256,-2.947,-46.067,179.875,5.949,149.101
C03021=1168.250,-2.698,-46.080,179.878,5.949,149.100
C03022=1168.245,-2.448,-46.093,179.881,5.949,149.099
C03023=1168.240,-2.199,-46.107,179.883,5.950,149.099
C03024=1168.235,-1.948,-46.121,179.885,5.951,149.098
C03025=1168.230,-1.700,-46.134,179.888,5.952,149.098
C03026=1168.224,-1.449,-46.148,179.890,5.952,149.097
C03027=1168.219,-1.200,-46.160,179.893,5.952,149.096
C03028=1168.214,-0.950,-46.175,179.895,5.953,149.096
C03029=1168.209,-0.701,-46.187,179.898,5.954,149.095
C03030=1168.204,-0.451,-46.201,179.900,5.955,149.095
C03031=1168.198,-0.202,-46.215,179.902,5.955,149.094
C03032=1168.194,0.048,-46.228,179.905,5.956,149.093
C03033=1168.188,0.297,-46.241,179.907,5.956,149.093
C03034=1168.184,0.547,-46.255,179.910,5.957,149.092
C03035=1168.178,0.796,-46.268,179.912,5.958,149.092
C03036=1168.173,1.046,-46.283,179.915,5.958,149.091
C03037=1168.168,1.295,-46.295,179.917,5.959,149.090
C03038=1168.163,1.545,-46.309,179.920,5.959,149.090
C03039=1168.157,1.815,-46.324,179.923,5.961,149.089
C03040=1168.152,2.084,-46.338,179.926,5.961,149.089
C03041=1168.147,2.353,-46.353,179.928,5.962,149.088
C03042=1168.141,2.622,-46.368,179.930,5.962,149.087
C03043=1168.135,2.872,-46.381,179.933,5.963,149.087
C03044=1168.131,3.121,-46.395,179.936,5.963,149.086
C03045=1168.126,3.372,-46.408,179.938,5.965,149.086
C03046=1168.120,3.621,-46.422,179.941,5.965,149.085
C03047=1168.116,3.870,-46.436,179.943,5.966,149.085
C03048=1168.110,4.120,-46.449,179.946,5.967,149.084
C03049=1168.105,4.370,-46.463,179.949,5.967,149.083
C03050=1168.100,4.619,-46.476,179.951,5.968,149.083
C03051=1168.095,4.869,-46.490,179.953,5.968,149.082
C03052=1168.090,5.118,-46.504,179.956,5.969,149.082
C03053=1168.085,5.368,-46.518,179.958,5.970,149.081
C03054=1168.080,5.617,-46.531,179.961,5.970,149.080
C03055=1168.075,5.867,-46.546,179.963,5.971,149.080
C03056=1168.069,6.117,-46.559,179.966,5.972,149.079
C03057=1168.065,6.366,-46.573,179.968,5.972,149.079
C03058=1168.060,6.615,-46.586,179.971,5.974,149.078
C03059=1168.054,6.865,-46.600,179.974,5.974,149.077
C03060=1168.049,7.115,-46.614,179.976,5.975,149.077
C03061=1168.044,7.364,-46.628,179.979,5.975,149.076
C03062=1168.039,7.614,-46.641,179.981,5.976,149.076
C03063=1168.034,7.864,-46.655,179.983,5.977,149.075
C03064=1168.029,8.113,-46.669,179.986,5.977,149.074
C03065=1168.024,8.363,-46.684,179.988,5.978,149.074
C03066=1168.019,8.613,-46.697,179.991,5.978,149.073
C03067=1168.014,8.862,-46.710,179.993,5.979,149.073
C03068=1168.009,9.111,-46.725,179.996,5.980,149.072
C03069=1168.004,9.361,-46.739,179.999,5.981,149.071
C03070=1167.998,9.611,-46.752,-179.999,5.982,149.071
C03071=1167.993,9.860,-46.766,-179.996,5.982,149.070
C03072=1167.988,10.110,-46.781,-179.994,5.983,149.070
C03073=1167.983,10.359,-46.794,-179.991,5.984,149.069
C03074=1167.978,10.608,-46.808,-179.989,5.984,149.068
C03075=1167.973,10.859,-46.822,-179.987,5.985,149.068
C03076=1167.968,11.108,-46.836,-179.984,5.985,149.067
C03077=1167.963,11.358,-46.850,-179.982,5.986,149.067
C03078=1167.958,11.607,-46.864,-179.979,5.987,149.066
C03079=1167.952,11.856,-46.878,-179.976,5.988,149.065
C03080=1167.948,12.106,-46.892,-179.974,5.989,149.065
C03081=1167.943,12.355,-46.906,-179.971,5.989,149.064
C03082=1167.938,12.606,-46.920,-179.969,5.990,149.064
C03083=1167.932,12.855,-46.934,-179.966,5.991,149.063
C03084=1167.927,13.104,-46.948,-179.964,5.991,149.063
C03085=1167.922,13.354,-46.962,-179.961,5.992,149.062
C03086=1167.917,13.603,-46.976,-179.958,5.993,149.061
C03087=1167.912,13.853,-46.990,-179.956,5.994,149.061
C03088=1167.907,14.103,-47.005,-179.953,5.994,149.060
C03089=1167.902,14.352,-47.019,-179.951,5.995,149.060
C03090=1167.896,14.601,-47.033,-179.949,5.996,149.059
C03091=1167.891,14.851,-47.047,-179.946,5.996,149.058
C03092=1167.886,15.101,-47.061,-179.944,5.997,149.058
C03093=1167.881,15.350,-47.076,-179.941,5.998,149.057
C03094=1167.876,15.599,-47.090,-179.938,5.999,149.057
C03095=1167.872,15.849,-47.103,-179.936,6.000,149.056
C03096=1167.867,16.099,-47.118,-179.934,6.000,149.055
C03097=1167.862,16.348,-47.132,-179.931,6.001,149.055
C03098=1167.857,16.598,-47.146,-179.928,6.001,149.054
C03099=1167.851,16.847,-47.160,-179.926,6.002,149.054
C03100=1167.846,17.097,-47.174,-179.923,6.003,149.053
C03101=1167.841,17.346,-47.189,-179.921,6.004,149.053
C03102=1167.836,17.596,-47.203,-179.918,6.005,149.052
C03103=1167.831,17.846,-47.218,-179.915,6.005,149.051
C03104=1167.825,18.095,-47.232,-179.913,6.006,149.051
C03105=1167.820,18.345,-47.246,-179.911,6.007,149.050
C03106=1167.815,18.595,-47.260,-179.908,6.007,149.050
C03107=1167.810,18.844,-47.275,-179.905,6.009,149.049
C03108=1167.805,19.094,-47.289,-179.903,6.010,149.048
C03109=1167.800,19.342,-47.303,-179.900,6.010,149.048
C03110=1167.795,19.592,-47.318,-179.898,6.011,149.047
C03111=1167.790,19.842,-47.332,-179.896,6.011,149.047
C03112=1167.785,20.091,-47.346,-179.893,6.012,149.046
C03113=1167.780,20.341,-47.361,-179.890,6.014,149.045
C03114=1167.775,20.591,-47.375,-179.887,6.014,149.045
C03115=1167.770,20.841,-47.389,-179.885,6.015,149.044
C03116=1167.765,21.089,-47.404,-179.883,6.015,149.044
C03117=1167.760,21.339,-47.418,-179.880,6.016,149.043
C03118=1167.754,21.589,-47.433,-179.878,6.017,149.042
C03119=1167.749,21.838,-47.447,-179.875,6.018,149.042
C03120=1167.744,22.088,-47.461,-179.872,6.019,149.041
C03121=1167.740,22.337,-47.476,-179.870,6.019,149.041
C03122=1167.735,22.587,-47.491,-179.867,6.020,149.040
C03123=1167.730,22.837,-47.505,-179.865,6.021,149.040
C03124=1167.724,23.086,-47.519,-179.862,6.021,149.039
C03125=1167.719,23.335,-47.534,-179.860,6.023,149.038
C03126=1167.714,23.585,-47.549,-179.857,6.023,149.038
C03127=1167.709,23.834,-47.563,-179.855,6.024,149.037
C03128=1167.704,24.084,-47.577,-179.852,6.024,149.037
C03129=1167.699,24.333,-47.592,-179.849,6.025,149.036
C03130=1167.695,24.583,-47.607,-179.847,6.027,149.035
C03131=1167.689,24.833,-47.621,-179.844,6.027,149.035
C03132=1167.684,25.082,-47.636,-179.842,6.028,149.034
C03133=1167.679,25.332,-47.651,-179.839,6.028,149.034
C03134=1167.674,25.582,-47.665,-179.837,6.029,149.033
C03135=1167.669,25.830,-47.680,-179.834,6.031,149.033
C03136=1167.663,26.080,-47.695,-179.831,6.031,149.032
C03137=1167.658,26.330,-47.709,-179.829,6.032,149.031
C03138=1167.654,26.579,-47.724,-179.826,6.032,149.031
C03139=1167.649,26.828,-47.738,-179.824,6.033,149.030
C03140=1167.643,27.078,-47.753,-179.821,6.034,149.030
C03141=1167.638,27.328,-47.768,-179.819,6.035,149.029
C03142=1167.633,27.577,-47.782,-179.816,6.036,149.028
C03143=1167.628,27.846,-47.798,-179.814,6.036,149.028
C03144=1167.622,28.115,-47.814,-179.811,6.038,149.027
C03145=1167.617,28.384,-47.830,-179.808,6.038,149.027
C03146=1167.611,28.653,-47.846,-179.805,6.040,149.026
C03147=1167.607,28.902,-47.861,-179.802,6.040,149.025
C03148=1167.602,29.152,-47.875,-179.800,6.041,149.025
C03149=1167.596,29.401,-47.891,-179.797,6.041,149.024
C03150=1167.592,29.651,-47.905,-179.795,6.042,149.024
C03151=1167.587,29.900,-47.920,-179.792,6.044,149.023
C03152=1167.581,30.150,-47.935,-179.790,6.044,149.023
C03153=1167.577,30.399,-47.950,-179.787,6.045,149.022
C03154=1167.572,30.649,-47.964,-179.785,6.046,149.021
C03155=1167.566,30.898,-47.980,-179.782,6.047,149.021
C03156=1167.561,31.148,-47.994,-179.779,6.048,149.020
C03157=1167.557,31.397,-48.009,-179.777,6.048,149.020
C03158=1167.551,31.647,-48.024,-179.774,6.049,149.019
C03159=1167.546,31.896,-48.039,-179.772,6.050,149.019
C03160=1167.541,32.146,-48.053,-179.769,6.051,149.018
C03161=1167.536,32.395,-48.069,-179.767,6.052,149.017
C03162=1167.531,32.645,-48.083,-179.764,6.052,149.017
C03163=1167.526,32.894,-48.099,-179.762,6.053,149.016
C03164=1167.521,33.144,-48.114,-179.759,6.055,149.016
C03165=1167.516,33.393,-48.128,-179.756,6.055,149.015
C03166=1167.511,33.643,-48.144,-179.754,6.056,149.014
C03167=1167.506,33.892,-48.159,-179.751,6.056,149.014
C03168=1167.500,34.142,-48.174,-179.749,6.058,149.013
C03169=1167.496,34.392,-48.189,-179.746,6.058,149.013
C03170=1167.491,34.642,-48.204,-179.744,6.059,149.012
C03171=1167.486,34.891,-48.219,-179.741,6.060,149.012
C03172=1167.481,35.140,-48.234,-179.738,6.061,149.011
C03173=1167.476,35.389,-48.249,-179.736,6.062,149.010
C03174=1167.471,35.639,-48.264,-179.733,6.062,149.010
C03175=1167.465,35.888,-48.279,-179.731,6.063,149.009
C03176=1167.461,36.137,-48.294,-179.728,6.065,149.009
C03177=1167.455,36.387,-48.309,-179.726,6.065,149.008
C03178=1167.450,36.636,-48.324,-179.723,6.066,149.008
C03179=1167.446,36.887,-48.340,-179.721,6.067,149.007
C03180=1167.441,37.136,-48.355,-179.718,6.068,149.006
C03181=1167.435,37.386,-48.370,-179.715,6.069,149.006
C03182=1167.431,37.635,-48.385,-179.713,6.069,149.005
C03183=1167.425,37.884,-48.401,-179.710,6.071,149.005
C03184=1167.421,38.133,-48.416,-179.707,6.072,149.004
C03185=1167.415,38.383,-48.430,-179.705,6.072,149.003
C03186=1167.410,38.632,-48.445,-179.703,6.073,149.003
C03187=1167.406,38.883,-48.461,-179.699,6.074,149.002
C03188=1167.400,39.132,-48.477,-179.697,6.075,149.002
C03189=1167.396,39.381,-48.492,-179.694,6.076,149.001
C03190=1167.390,39.631,-48.507,-179.692,6.077,149.001
C03191=1167.385,39.880,-48.522,-179.689,6.078,149.000
C03192=1167.380,40.130,-48.537,-179.687,6.079,149.000
C03193=1167.376,40.379,-48.553,-179.684,6.079,148.999
C03194=1167.370,40.629,-48.568,-179.682,6.081,148.999
C03195=1167.365,40.878,-48.584,-179.679,6.081,148.998
C03196=1167.360,41.127,-48.599,-179.677,6.082,148.997
C03197=1167.355,41.377,-48.615,-179.674,6.083,148.997
C03198=1167.350,41.626,-48.630,-179.671,6.084,148.996
C03199=1167.345,41.876,-48.645,-179.669,6.085,148.996
C03200=1167.340,42.126,-48.660,-179.666,6.085,148.995
C03201=1167.335,42.375,-48.675,-179.663,6.087,148.995
C03202=1167.330,42.624,-48.691,-179.661,6.087,148.994
C03203=1167.325,42.874,-48.707,-179.659,6.088,148.993
C03204=1167.320,43.124,-48.722,-179.655,6.090,148.993
C03205=1167.315,43.373,-48.737,-179.653,6.090,148.992
C03206=1167.310,43.622,-48.753,-179.651,6.091,148.992
C03207=1167.305,43.871,-48.768,-179.648,6.093,148.991
C03208=1167.300,44.122,-48.784,-179.645,6.093,148.990
C03209=1167.295,44.371,-48.800,-179.643,6.094,148.990
C03210=1167.290,44.620,-48.815,-179.640,6.094,148.989
C03211=1167.285,44.869,-48.830,-179.638,6.096,148.989
C03212=1167.280,45.120,-48.846,-179.635,6.097,148.988
C03213=1167.275,45.369,-48.862,-179.633,6.097,148.988
C03214=1167.270,45.618,-48.877,-179.630,6.099,148.987
C03215=1167.264,45.867,-48.892,-179.627,6.100,148.987
C03216=1167.260,46.118,-48.908,-179.625,6.100,148.986
C03217=1167.255,46.366,-48.924,-179.622,6.102,148.986
C03218=1167.250,46.615,-48.940,-179.619,6.102,148.985
C03219=1167.245,46.865,-48.956,-179.617,6.103,148.984
C03220=1167.240,47.115,-48.971,-179.614,6.104,148.984
C03221=1167.235,47.364,-48.986,-179.611,6.105,148.983
C03222=1167.230,47.613,-49.002,-179.609,6.106,148.983
C03223=1167.225,47.863,-49.018,-179.606,6.107,148.982
C03224=1167.220,48.113,-49.033,-179.604,6.108,148.982
C03225=1167.215,48.362,-49.050,-179.601,6.108,148.981
C03226=1167.210,48.611,-49.065,-179.598,6.110,148.980
C03227=1167.205,48.861,-49.080,-179.596,6.111,148.980
C03228=1167.200,49.110,-49.096,-179.594,6.111,148.979
C03229=1167.195,49.360,-49.112,-179.590,6.113,148.979
C03230=1167.190,49.610,-49.128,-179.588,6.114,148.978
C03231=1167.185,49.858,-49.143,-179.586,6.114,148.978
C03232=1167.180,50.108,-49.159,-179.583,6.116,148.977
C03233=1167.175,50.358,-49.175,-179.580,6.116,148.976
C03234=1167.170,50.607,-49.190,-179.578,6.117,148.976
C03235=1167.165,50.857,-49.207,-179.575,6.118,148.975
C03236=1167.160,51.106,-49.223,-179.573,6.119,148.975
C03237=1167.155,51.355,-49.238,-179.569,6.121,148.974
C03238=1167.150,51.605,-49.254,-179.567,6.121,148.974
C03239=1167.145,51.854,-49.270,-179.565,6.122,148.973
C03240=1167.140,52.104,-49.286,-179.562,6.124,148.973
C03241=1167.135,52.354,-49.301,-179.559,6.124,148.972
C03242=1167.130,52.602,-49.318,-179.557,6.125,148.972
C03243=1167.125,52.852,-49.334,-179.554,6.126,148.971
C03244=1167.120,53.102,-49.349,-179.552,6.127,148.970
C03245=1167.115,53.351,-49.366,-179.549,6.128,148.970
C03246=1167.110,53.601,-49.382,-179.546,6.129,148.969
C03247=1167.104,53.869,-49.399,-179.544,6.130,148.969
C03248=1167.099,54.138,-49.416,-179.541,6.131,148.968
C03249=1167.094,54.407,-49.433,-179.538,6.132,148.968
C03250=1167.089,54.675,-49.451,-179.535,6.133,148.967
C03251=1167.083,54.924,-49.466,-179.533,6.134,148.967
C03252=1167.078,55.174,-49.482,-179.530,6.135,148.966
C03253=1167.073,55.423,-49.499,-179.528,6.136,148.965
C03254=1167.069,55.673,-49.515,-179.524,6.138,148.965
C03255=1167.064,55.922,-49.530,-179.522,6.139,148.964
C03256=1167.059,56.171,-49.546,-179.520,6.139,148.964
C03257=1167.054,56.420,-49.562,-179.517,6.141,148.963
C03258=1167.048,56.670,-49.579,-179.514,6.141,148.963
C03259=1167.043,56.920,-49.595,-179.511,6.143,148.962
C03260=1167.038,57.169,-49.611,-179.509,6.143,148.961
C03261=1167.034,57.419,-49.627,-179.507,6.144,148.961
C03262=1167.029,57.668,-49.643,-179.503,6.146,148.960
C03263=1167.024,57.918,-49.659,-179.501,6.146,148.960
C03264=1167.019,58.167,-49.675,-179.498,6.148,148.959
C03265=1167.014,58.416,-49.692,-179.496,6.149,148.959
C03266=1167.009,58.666,-49.708,-179.493,6.149,148.958
C03267=1167.004,58.915,-49.724,-179.491,6.151,148.958
C03268=1166.999,59.165,-49.740,-179.488,6.151,148.957
C03269=1166.994,59.414,-49.757,-179.485,6.153,148.957
C03270=1166.989,59.663,-49.772,-179.483,6.153,148.956
C03271=1166.985,59.913,-49.789,-179.480,6.154,148.955
C03272=1166.979,60.162,-49.805,-179.477,6.156,148.955
C03273=1166.975,60.412,-49.821,-179.475,6.157,148.954
C03274=1166.969,60.661,-49.838,-179.472,6.158,148.954
C03275=1166.964,60.911,-49.854,-179.470,6.159,148.953
C03276=1166.959,61.160,-49.870,-179.467,6.159,148.953
C03277=1166.955,61.409,-49.887,-179.464,6.161,148.952
C03278=1166.949,61.659,-49.903,-179.462,6.161,148.952
C03279=1166.945,61.908,-49.919,-179.459,6.163,148.951
C03280=1166.940,62.157,-49.936,-179.457,6.164,148.951
C03281=1166.935,62.407,-49.951,-179.454,6.165,148.950
C03282=1166.930,62.657,-49.969,-179.451,6.166,148.950
C03283=1166.924,62.906,-49.985,-179.449,6.167,148.949
C03284=1166.920,63.156,-50.001,-179.446,6.168,148.948
C03285=1166.915,63.405,-50.017,-179.443,6.169,148.948
C03286=1166.910,63.654,-50.034,-179.441,6.171,148.947
C03287=1166.904,63.903,-50.051,-179.438,6.171,148.947
C03288=1166.900,64.153,-50.067,-179.435,6.173,148.946
C03289=1166.895,64.403,-50.084,-179.433,6.173,148.946
C03290=1166.890,64.651,-50.100,-179.430,6.174,148.945
C03291=1166.886,64.901,-50.116,-179.427,6.175,148.945
C03292=1166.880,65.150,-50.133,-179.425,6.176,148.944
C03293=1166.875,65.400,-50.149,-179.422,6.178,148.944
C03294=1166.870,65.650,-50.166,-179.420,6.178,148.943
C03295=1166.865,65.898,-50.182,-179.417,6.180,148.943
C03296=1166.860,66.148,-50.200,-179.414,6.181,148.942
C03297=1166.855,66.397,-50.216,-179.412,6.182,148.941
C03298=1166.850,66.647,-50.232,-179.409,6.183,148.941
C03299=1166.846,66.897,-50.248,-179.406,6.185,148.940
C03300=1166.840,67.146,-50.265,-179.404,6.185,148.940
C03301=1166.835,67.395,-50.282,-179.402,6.186,148.939
C03302=1166.831,67.645,-50.299,-179.398,6.187,148.939
C03303=1166.826,67.893,-50.315,-179.396,6.188,148.938
C03304=1166.821,68.143,-50.332,-179.393,6.190,148.938
C03305=1166.816,68.393,-50.349,-179.391,6.190,148.937
C03306=1166.811,68.642,-50.365,-179.388,6.192,148.937
C03307=1166.806,68.891,-50.383,-179.385,6.193,148.936
C03308=1166.801,69.141,-50.398,-179.383,6.194,148.936
C03309=1166.796,69.390,-50.415,-179.380,6.195,148.935
C03310=1166.791,69.640,-50.432,-179.377,6.196,148.934
C03311=1166.786,69.889,-50.449,-179.375,6.197,148.934
C03312=1166.781,70.138,-50.465,-179.372,6.199,148.933
C03313=1166.776,70.388,-50.482,-179.370,6.199,148.933
C03314=1166.772,70.638,-50.499,-179.367,6.201,148.932
C03315=1166.766,70.887,-50.516,-179.364,6.202,148.932
C03316=1166.761,71.136,-50.533,-179.361,6.203,148.931
C03317=1166.757,71.386,-50.549,-179.359,6.204,148.931
C03318=1166.752,71.635,-50.566,-179.356,6.204,148.930
C03319=1166.746,71.884,-50.583,-179.354,6.206,148.930
C03320=1166.742,72.133,-50.601,-179.351,6.207,148.929
C03321=1166.737,72.383,-50.617,-179.348,6.208,148.929
C03322=1166.732,72.632,-50.634,-179.346,6.209,148.928
C03323=1166.727,72.881,-50.651,-179.343,6.210,148.928
C03324=1166.722,73.131,-50.668,-179.341,6.211,148.927
C03325=1166.717,73.381,-50.685,-179.338,6.213,148.926
C03326=1166.712,73.629,-50.701,-179.335,6.214,148.926
C03327=1166.707,73.879,-50.718,-179.332,6.215,148.925
C03328=1166.702,74.129,-50.735,-179.330,6.216,148.925
C03329=1166.697,74.379,-50.752,-179.327,6.217,148.924
C03330=1166.692,74.627,-50.769,-179.325,6.218,148.924
C03331=1166.687,74.877,-50.787,-179.322,6.220,148.923
C03332=1166.683,75.126,-50.803,-179.319,6.220,148.923
C03333=1166.677,75.376,-50.821,-179.317,6.222,148.922
C03334=1166.673,75.625,-50.837,-179.314,6.224,148.922
C03335=1166.667,75.874,-50.855,-179.311,6.224,148.921
C03336=1166.663,76.123,-50.872,-179.309,6.226,148.921
C03337=1166.658,76.373,-50.889,-179.306,6.226,148.920
C03338=1166.653,76.623,-50.906,-179.303,6.228,148.920
C03339=1166.648,76.872,-50.923,-179.301,6.228,148.919
C03340=1166.643,77.120,-50.940,-179.298,6.230,148.919
C03341=1166.638,77.370,-50.957,-179.296,6.231,148.918
C03342=1166.634,77.620,-50.974,-179.292,6.232,148.918
C03343=1166.629,77.869,-50.992,-179.290,6.233,148.917
C03344=1166.623,78.119,-51.009,-179.287,6.235,148.916
C03345=1166.618,78.368,-51.025,-179.285,6.235,148.916
C03346=1166.613,78.617,-51.043,-179.282,6.237,148.916
C03347=1166.609,78.866,-51.060,-179.280,6.238,148.915
C03348=1166.604,79.116,-51.077,-179.277,6.239,148.915
C03349=1166.599,79.366,-51.094,-179.274,6.240,148.914
C03350=1166.594,79.615,-51.112,-179.272,6.242,148.913
C03351=1166.588,79.883,-51.130,-179.268,6.243,148.913
C03352=1166.583,80.152,-51.149,-179.266,6.244,148.912
C03353=1166.579,80.420,-51.168,-179.263,6.245,148.912
C03354=1166.573,80.688,-51.186,-179.260,6.247,148.911
C03355=1166.567,80.938,-51.203,-179.258,6.247,148.911
C03356=1166.563,81.186,-51.221,-179.255,6.249,148.910
C03357=1166.558,81.436,-51.238,-179.252,6.250,148.910
C03358=1166.553,81.686,-51.255,-179.249,6.251,148.909
C03359=1166.549,81.935,-51.273,-179.247,6.253,148.909
C03360=1166.543,82.185,-51.290,-179.244,6.253,148.908
C03361=1166.538,82.434,-51.308,-179.241,6.255,148.908
C03362=1166.533,82.683,-51.325,-179.239,6.256,148.907
C03363=1166.529,82.932,-51.342,-179.236,6.257,148.907
C03364=1166.523,83.182,-51.359,-179.234,6.258,148.906
C03365=1166.518,83.431,-51.377,-179.231,6.260,148.905
C03366=1166.514,83.680,-51.394,-179.228,6.261,148.905
C03367=1166.509,83.929,-51.412,-179.226,6.262,148.905
C03368=1166.504,84.179,-51.429,-179.223,6.264,148.904
C03369=1166.499,84.428,-51.447,-179.220,6.264,148.904
C03370=1166.494,84.678,-51.464,-179.217,6.266,148.903
C03371=1166.489,84.927,-51.482,-179.215,6.267,148.902
C03372=1166.485,85.176,-51.500,-179.212,6.268,148.902
C03373=1166.479,85.426,-51.517,-179.209,6.270,148.901
C03374=1166.475,85.675,-51.535,-179.207,6.271,148.901
C03375=1166.470,85.925,-51.552,-179.204,6.272,148.901
C03376=1166.465,86.174,-51.570,-179.202,6.273,148.900
C03377=1166.460,86.423,-51.588,-179.199,6.274,148.900
C03378=1166.455,86.673,-51.605,-179.196,6.276,148.899
C03379=1166.451,86.922,-51.622,-179.194,6.277,148.898
C03380=1166.446,87.172,-51.640,-179.191,6.278,148.898
C03381=1166.441,87.421,-51.658,-179.188,6.279,148.897
C03382=1166.436,87.670,-51.676,-179.186,6.281,148.897
C03383=1166.431,87.919,-51.694,-179.183,6.282,148.897
C03384=1166.426,88.169,-51.711,-179.180,6.283,148.896
C03385=1166.421,88.418,-51.729,-179.177,6.285,148.895
C03386=1166.416,88.667,-51.746,-179.175,6.285,148.895
C03387=1166.411,88.917,-51.763,-179.172,6.287,148.894
C03388=1166.406,89.166,-51.781,-179.169,6.288,148.894
C03389=1166.401,89.415,-51.799,-179.167,6.289,148.893
C03390=1166.397,89.664,-51.817,-179.164,6.291,148.893
C03391=1166.391,89.914,-51.835,-179.162,6.292,148.892
C03392=1166.386,90.163,-51.853,-179.159,6.293,148.892
C03393=1166.381,90.412,-51.871,-179.156,6.295,148.891
C03394=1166.377,90.662,-51.889,-179.154,6.296,148.891
C03395=1166.371,90.911,-51.906,-179.151,6.297,148.890
C03396=1166.367,91.160,-51.923,-179.148,6.298,148.890
C03397=1166.362,91.409,-51.941,-179.146,6.299,148.890
C03398=1166.357,91.659,-51.959,-179.143,6.301,148.889
C03399=1166.352,91.908,-51.977,-179.140,6.302,148.888
C03400=1166.348,92.157,-51.995,-179.138,6.303,148.888
C03401=1166.342,92.407,-52.012,-179.134,6.305,148.887
C03402=1166.338,92.657,-52.031,-179.132,6.306,148.887
C03403=1166.333,92.906,-52.049,-179.130,6.307,148.887
C03404=1166.328,93.155,-52.067,-179.127,6.308,148.886
C03405=1166.323,93.404,-52.085,-179.124,6.310,148.885
C03406=1166.318,93.653,-52.103,-179.122,6.311,148.885
C03407=1166.313,93.902,-52.121,-179.119,6.312,148.884
C03408=1166.309,94.152,-52.139,-179.116,6.313,148.884
C03409=1166.304,94.401,-52.157,-179.113,6.315,148.884
C03410=1166.299,94.650,-52.175,-179.111,6.316,148.883
C03411=1166.294,94.900,-52.193,-179.108,6.317,148.883
C03412=1166.289,95.149,-52.211,-179.105,6.319,148.882
C03413=1166.285,95.398,-52.229,-179.103,6.320,148.881
C03414=1166.280,95.647,-52.247,-179.100,6.321,148.881
C03415=1166.274,95.897,-52.266,-179.098,6.322,148.881
C03416=1166.269,96.146,-52.283,-179.095,6.324,148.880
C03417=1166.264,96.395,-52.301,-179.092,6.325,148.880
C03418=1166.260,96.645,-52.320,-179.090,6.326,148.879
C03419=1166.255,96.894,-52.338,-179.087,6.328,148.878
C03420=1166.250,97.143,-52.356,-179.084,6.329,148.878
C03421=1166.245,97.393,-52.374,-179.082,6.330,148.878
C03422=1166.240,97.642,-52.392,-179.079,6.331,148.877
C03423=1166.235,97.891,-52.410,-179.076,6.333,148.877
C03424=1166.231,98.141,-52.428,-179.074,6.334,148.876
C03425=1166.225,98.390,-52.447,-179.071,6.335,148.876
C03426=1166.220,98.640,-52.465,-179.068,6.337,148.875
C03427=1166.216,98.889,-52.483,-179.066,6.338,148.875
C03428=1166.211,99.138,-52.501,-179.062,6.339,148.874
C03429=1166.207,99.387,-52.520,-179.060,6.341,148.874
C03430=1166.202,99.636,-52.538,-179.058,6.342,148.873
C03431=1166.196,99.886,-52.556,-179.054,6.343,148.873
C03432=1166.191,100.135,-52.574,-179.052,6.345,148.872
C03433=1166.186,100.384,-52.592,-179.050,6.346,148.872
C03434=1166.182,100.633,-52.611,-179.047,6.348,148.871
C03435=1166.177,100.883,-52.629,-179.044,6.349,148.871
C03436=1166.172,101.132,-52.648,-179.041,6.351,148.870
C03437=1166.167,101.381,-52.666,-179.039,6.352,148.870
C03438=1166.162,101.631,-52.684,-179.036,6.353,148.869
C03439=1166.158,101.880,-52.703,-179.033,6.355,148.869
C03440=1166.153,102.129,-52.721,-179.031,6.356,148.868
C03441=1166.147,102.378,-52.739,-179.027,6.357,148.868
C03442=1166.143,102.628,-52.758,-179.025,6.359,148.867
C03443=1166.138,102.877,-52.776,-179.023,6.360,148.867
C03444=1166.133,103.126,-52.795,-179.020,6.361,148.867
C03445=1166.128,103.376,-52.813,-179.017,6.363,148.866
C03446=1166.124,103.625,-52.832,-179.014,6.364,148.866
C03447=1166.119,103.874,-52.850,-179.012,6.365,148.865
C03448=1166.113,104.123,-52.869,-179.009,6.367,148.864
C03449=1166.109,104.373,-52.888,-179.006,6.368,148.864
C03450=1166.104,104.622,-52.906,-179.004,6.369,148.864
C03451=1166.099,104.871,-52.924,-179.001,6.371,148.863
C03452=1166.095,105.121,-52.943,-178.998,6.372,148.863
C03453=1166.090,105.370,-52.961,-178.996,6.373,148.862
C03454=1166.084,105.619,-52.980,-178.993,6.375,148.862
C03455=1166.080,105.888,-53.000,-178.990,6.376,148.861
C03456=1166.074,106.156,-53.020,-178.987,6.378,148.861
C03457=1166.069,106.424,-53.040,-178.984,6.379,148.860
C03458=1166.063,106.692,-53.060,-178.981,6.381,148.860
C03459=1166.059,106.942,-53.079,-178.978,6.383,148.859
C03460=1166.055,107.191,-53.097,-178.976,6.383,148.859
C03461=1166.049,107.440,-53.116,-178.973,6.385,148.858
C03462=1166.045,107.689,-53.135,-178.970,6.387,148.858
C03463=1166.039,107.939,-53.154,-178.968,6.388,148.857
C03464=1166.035,108.187,-53.172,-178.965,6.389,148.857
C03465=1166.030,108.438,-53.191,-178.962,6.391,148.856
C03466=1166.025,108.686,-53.210,-178.960,6.392,148.856
C03467=1166.021,108.936,-53.228,-178.957,6.394,148.856
C03468=1166.015,109.185,-53.248,-178.954,6.395,148.855
C03469=1166.010,109.434,-53.266,-178.952,6.396,148.854
C03470=1166.006,109.684,-53.285,-178.949,6.398,148.854
C03471=1166.001,109.932,-53.304,-178.946,6.400,148.854
C03472=1165.996,110.182,-53.323,-178.944,6.400,148.853
C03473=1165.991,110.431,-53.342,-178.941,6.402,148.853
C03474=1165.986,110.681,-53.360,-178.938,6.404,148.852
C03475=1165.982,110.930,-53.379,-178.935,6.405,148.852
C03476=1165.976,111.179,-53.399,-178.933,6.406,148.851
C03477=1165.972,111.429,-53.417,-178.930,6.408,148.851
C03478=1165.967,111.677,-53.436,-178.927,6.409,148.850
C03479=1165.963,111.927,-53.455,-178.925,6.411,148.850
C03480=1165.957,112.176,-53.474,-178.922,6.412,148.849
C03481=1165.953,112.425,-53.492,-178.919,6.413,148.849
C03482=1165.948,112.674,-53.512,-178.917,6.415,148.849
C03483=1165.943,112.923,-53.530,-178.914,6.417,148.848
C03484=1165.938,113.173,-53.550,-178.911,6.417,148.847
C03485=1165.934,113.422,-53.568,-178.909,6.419,148.847
C03486=1165.928,113.672,-53.587,-178.906,6.421,148.847
C03487=1165.923,113.921,-53.607,-178.903,6.422,148.846
C03488=1165.919,114.170,-53.626,-178.901,6.423,148.846
C03489=1165.914,114.419,-53.645,-178.898,6.425,148.845
C03490=1165.910,114.668,-53.664,-178.895,6.426,148.845
C03491=1165.904,114.917,-53.683,-178.892,6.428,148.844
C03492=1165.899,115.167,-53.702,-178.890,6.430,148.844
C03493=1165.895,115.416,-53.721,-178.887,6.430,148.843
C03494=1165.890,115.665,-53.741,-178.884,6.432,148.843
C03495=1165.885,115.914,-53.760,-178.882,6.434,148.843
C03496=1165.880,116.164,-53.778,-178.879,6.436,148.842
C03497=1165.875,116.413,-53.798,-178.876,6.437,148.842
C03498=1165.870,116.662,-53.817,-178.874,6.438,148.841
C03499=1165.866,116.911,-53.836,-178.871,6.440,148.841
C03500=1165.861,117.160,-53.856,-178.868,6.441,148.840
C03501=1165.856,117.409,-53.875,-178.865,6.443,148.840
C03502=1165.852,117.659,-53.894,-178.862,6.444,148.839
C03503=1165.846,117.907,-53.913,-178.860,6.445,148.839
C03504=1165.841,118.158,-53.932,-178.857,6.447,148.838
C03505=1165.837,118.407,-53.951,-178.855,6.449,148.838
C03506=1165.832,118.656,-53.971,-178.852,6.450,148.838
C03507=1165.827,118.905,-53.990,-178.849,6.452,148.837
C03508=1165.822,119.154,-54.010,-178.847,6.453,148.837
C03509=1165.818,119.403,-54.029,-178.844,6.454,148.836
C03510=1165.812,119.652,-54.048,-178.841,6.456,148.836
C03511=1165.808,119.902,-54.068,-178.839,6.458,148.835
C03512=1165.803,120.151,-54.087,-178.835,6.459,148.835
C03513=1165.798,120.400,-54.106,-178.833,6.460,148.834
C03514=1165.794,120.650,-54.126,-178.830,6.462,148.834
C03515=1165.788,120.898,-54.145,-178.828,6.464,148.834
C03516=1165.783,121.148,-54.164,-178.825,6.465,148.833
C03517=1165.779,121.397,-54.184,-178.822,6.467,148.833
C03518=1165.774,121.646,-54.204,-178.819,6.468,148.832
C03519=1165.770,121.895,-54.223,-178.817,6.469,148.832
C03520=1165.765,122.145,-54.243,-178.814,6.471,148.831
C03521=1165.760,122.394,-54.262,-178.812,6.473,148.831
C03522=1165.756,122.643,-54.281,-178.809,6.474,148.831
C03523=1165.750,122.892,-54.300,-178.806,6.476,148.830
C03524=1165.746,123.141,-54.320,-178.803,6.478,148.830
C03525=1165.741,123.391,-54.340,-178.801,6.478,148.829
C03526=1165.736,123.639,-54.360,-178.798,6.480,148.829
C03527=1165.731,123.889,-54.379,-178.795,6.482,148.828
C03528=1165.726,124.138,-54.399,-178.792,6.483,148.828
C03529=1165.722,124.387,-54.418,-178.790,6.485,148.827
C03530=1165.717,124.636,-54.437,-178.787,6.487,148.827
C03531=1165.712,124.886,-54.457,-178.784,6.488,148.827
C03532=1165.708,125.135,-54.478,-178.782,6.489,148.826
C03533=1165.702,125.384,-54.497,-178.779,6.491,148.826
C03534=1165.698,125.633,-54.516,-178.776,6.492,148.825
C03535=1165.693,125.883,-54.536,-178.773,6.494,148.825
C03536=1165.688,126.131,-54.556,-178.771,6.496,148.824
C03537=1165.683,126.381,-54.576,-178.768,6.498,148.824
C03538=1165.678,126.630,-54.595,-178.765,6.499,148.824
C03539=1165.673,126.878,-54.615,-178.763,6.500,148.823
C03540=1165.669,127.128,-54.635,-178.760,6.502,148.823
C03541=1165.664,127.378,-54.655,-178.757,6.503,148.822
C03542=1165.659,127.627,-54.674,-178.755,6.505,148.822
C03543=1165.655,127.875,-54.694,-178.752,6.507,148.821
C03544=1165.650,128.125,-54.713,-178.749,6.509,148.821
C03545=1165.646,128.374,-54.734,-178.746,6.510,148.821
C03546=1165.641,128.623,-54.754,-178.744,6.512,148.820
C03547=1165.636,128.872,-54.773,-178.742,6.513,148.820
C03548=1165.630,129.121,-54.794,-178.738,6.514,148.819
C03549=1165.626,129.371,-54.813,-178.736,6.516,148.819
C03550=1165.621,129.620,-54.834,-178.733,6.518,148.818
C03551=1165.616,129.869,-54.853,-178.730,6.519,148.818
C03552=1165.611,130.118,-54.873,-178.728,6.521,148.818
C03553=1165.607,130.367,-54.893,-178.725,6.523,148.817
C03554=1165.602,130.617,-54.913,-178.722,6.525,148.817
C03555=1165.597,130.866,-54.933,-178.719,6.526,148.816
C03556=1165.592,131.115,-54.952,-178.717,6.527,148.816
C03557=1165.588,131.364,-54.973,-178.714,6.529,148.815
C03558=1165.583,131.613,-54.992,-178.711,6.530,148.815
C03559=1165.578,131.881,-55.015,-178.709,6.532,148.815
C03560=1165.573,132.150,-55.036,-178.706,6.534,148.814
C03561=1165.567,132.419,-55.058,-178.702,6.536,148.814
C03562=1165.562,132.687,-55.079,-178.700,6.538,148.813
C03563=1165.558,132.937,-55.099,-178.697,6.540,148.813
C03564=1165.553,133.186,-55.119,-178.694,6.541,148.812
C03565=1165.548,133.434,-55.139,-178.692,6.542,148.812
C03566=1165.543,133.684,-55.160,-178.689,6.544,148.811
C03567=1165.538,133.933,-55.179,-178.686,6.545,148.811
C03568=1165.534,134.182,-55.200,-178.683,6.547,148.811
C03569=1165.529,134.431,-55.220,-178.681,6.549,148.810
C03570=1165.524,134.681,-55.240,-178.678,6.550,148.810
C03571=1165.520,134.930,-55.260,-178.675,6.552,148.809
C03572=1165.515,135.179,-55.281,-178.673,6.554,148.809
C03573=1165.509,135.428,-55.300,-178.670,6.556,148.809
C03574=1165.505,135.677,-55.321,-178.667,6.557,148.808
C03575=1165.501,135.926,-55.341,-178.664,6.559,148.808
C03576=1165.495,136.176,-55.361,-178.661,6.560,148.807
C03577=1165.491,136.425,-55.382,-178.659,6.562,148.807
C03578=1165.486,136.674,-55.402,-178.656,6.564,148.806
C03579=1165.482,136.922,-55.422,-178.654,6.565,148.806
C03580=1165.476,137.172,-55.443,-178.651,6.567,148.806
C03581=1165.472,137.421,-55.463,-178.648,6.568,148.805
C03582=1165.467,137.670,-55.483,-178.646,6.570,148.805
C03583=1165.462,137.918,-55.504,-178.643,6.572,148.804
C03584=1165.457,138.168,-55.524,-178.640,6.574,148.804
C03585=1165.452,138.417,-55.544,-178.638,6.575,148.804
C03586=1165.448,138.666,-55.564,-178.635,6.577,148.803
C03587=1165.443,138.916,-55.585,-178.632,6.578,148.803
C03588=1165.438,139.164,-55.606,-178.629,6.580,148.802
C03589=1165.434,139.414,-55.625,-178.626,6.582,148.802
C03590=1165.428,139.663,-55.646,-178.624,6.584,148.802
C03591=1165.424,139.912,-55.667,-178.621,6.585,148.801
C03592=1165.420,140.161,-55.687,-178.618,6.587,148.801
C03593=1165.414,140.410,-55.708,-178.615,6.589,148.800
C03594=1165.410,140.659,-55.729,-178.613,6.591,148.800
C03595=1165.406,140.908,-55.749,-178.610,6.592,148.800
C03596=1165.400,141.158,-55.770,-178.607,6.594,148.799
C03597=1165.396,141.407,-55.790,-178.605,6.596,148.799
C03598=1165.391,141.656,-55.810,-178.602,6.597,148.798
C03599=1165.386,141.905,-55.831,-178.599,6.599,148.798
C03600=1165.382,142.154,-55.851,-178.596,6.601,148.798
C03601=1165.376,142.404,-55.872,-178.594,6.603,148.797
C03602=1165.372,142.653,-55.893,-178.591,6.604,148.797
C03603=1165.368,142.902,-55.913,-178.588,6.606,148.796
C03604=1165.362,143.151,-55.934,-178.585,6.608,148.796
C03605=1165.358,143.400,-55.954,-178.583,6.608,148.796
C03606=1165.353,143.649,-55.975,-178.580,6.610,148.795
C03607=1165.348,143.898,-55.996,-178.578,6.612,148.795
C03608=1165.343,144.147,-56.017,-178.575,6.614,148.794
C03609=1165.339,144.396,-56.038,-178.572,6.615,148.794
C03610=1165.334,144.645,-56.059,-178.570,6.617,148.794
C03611=1165.330,144.894,-56.079,-178.567,6.619,148.793
C03612=1165.325,145.144,-56.100,-178.564,6.621,148.793
C03613=1165.320,145.393,-56.121,-178.561,6.622,148.792
C03614=1165.315,145.642,-56.142,-178.559,6.624,148.792
C03615=1165.311,145.891,-56.162,-178.556,6.626,148.792
C03616=1165.306,146.140,-56.183,-178.553,6.628,148.791
C03617=1165.301,146.389,-56.203,-178.551,6.629,148.791
C03618=1165.296,146.638,-56.225,-178.548,6.631,148.791
C03619=1165.292,146.887,-56.245,-178.545,6.633,148.790
C03620=1165.287,147.136,-56.266,-178.543,6.635,148.790
C03621=1165.282,147.385,-56.287,-178.540,6.636,148.789
C03622=1165.277,147.634,-56.308,-178.537,6.639,148.789
C03623=1165.273,147.883,-56.330,-178.534,6.641,148.789
C03624=1165.268,148.132,-56.350,-178.531,6.642,148.788
C03625=1165.263,148.382,-56.371,-178.529,6.644,148.788
C03626=1165.259,148.631,-56.392,-178.526,6.646,148.787
C03627=1165.254,148.879,-56.413,-178.523,6.648,148.787
C03628=1165.249,149.129,-56.434,-178.520,6.649,148.787
C03629=1165.244,149.377,-56.455,-178.518,6.651,148.786
C03630=1165.240,149.627,-56.476,-178.515,6.653,148.786
C03631=1165.236,149.876,-56.497,-178.512,6.654,148.786
C03632=1165.230,150.125,-56.518,-178.510,6.656,148.785
C03633=1165.225,150.374,-56.539,-178.507,6.658,148.785
C03634=1165.221,150.623,-56.560,-178.504,6.660,148.784
C03635=1165.216,150.872,-56.581,-178.502,6.661,148.784
C03636=1165.211,151.122,-56.602,-178.499,6.663,148.784
C03637=1165.206,151.370,-56.624,-178.496,6.665,148.783
C03638=1165.202,151.619,-56.644,-178.493,6.667,148.783
C03639=1165.197,151.868,-56.666,-178.491,6.668,148.783
C03640=1165.192,152.117,-56.687,-178.488,6.670,148.782
C03641=1165.188,152.367,-56.708,-178.485,6.672,148.782
C03642=1165.183,152.616,-56.729,-178.483,6.674,148.781
C03643=1165.178,152.865,-56.750,-178.480,6.675,148.781
C03644=1165.173,153.113,-56.772,-178.477,6.677,148.781
C03645=1165.169,153.362,-56.792,-178.475,6.679,148.780
C03646=1165.165,153.612,-56.814,-178.472,6.681,148.780
C03647=1165.159,153.861,-56.835,-178.469,6.682,148.780
C03648=1165.154,154.110,-56.857,-178.466,6.685,148.779
C03649=1165.150,154.359,-56.878,-178.463,6.687,148.779
C03650=1165.146,154.608,-56.900,-178.460,6.688,148.778
C03651=1165.141,154.857,-56.921,-178.458,6.690,148.778
C03652=1165.136,155.106,-56.942,-178.455,6.692,148.778
C03653=1165.131,155.355,-56.963,-178.452,6.694,148.777
C03654=1165.127,155.604,-56.985,-178.450,6.695,148.777
C03655=1165.122,155.853,-57.006,-178.447,6.697,148.777
C03656=1165.117,156.102,-57.027,-178.444,6.699,148.776
C03657=1165.112,156.351,-57.049,-178.442,6.701,148.776
C03658=1165.108,156.601,-57.070,-178.439,6.702,148.775
C03659=1165.103,156.849,-57.092,-178.436,6.704,148.775
C03660=1165.098,157.098,-57.112,-178.434,6.706,148.775
